(* CODESYS project mobject-server.library
   Company: mobject
   DefaultNamespace: mobject-server
   Version: 0.10.0
   Placeholder: mobject-server
   Author: mobject dev team
   Title: mobject-server

Project tree, tasks and I/O mapping:
  libraries: mobject-core, 0.3.0 (mobject); Tc2_Standard, * (Beckhoff Automation GmbH); Tc2_System, * (Beckhoff Automation GmbH); Tc2_Utilities, * (Beckhoff Automation GmbH)
  _Internal/
    AsyncResponse/
      HeaderAccessor/
        interface I_AsyncResponseHeaderAccessor: TryGetResponseIdFromRequest, TryGetSessionIdFromRequest, TryGetSessionIdFromResponse
      Manager/
        function block AsyncResponseManager [ST]: FB_init, CreateAsyncResponseSessionData, CreateAsyncResponseSessionDataProxy, TryConvertResponseToAsyncResponseSessionData, TryHandleIncomingRequest
        interface I_AsyncResponseManager: TryConvertResponseToAsyncResponseSessionData, TryHandleIncomingRequest
      Middleware/
        function block AsyncResponseMiddleware [ST]: FB_init, Handle
      Proxy/
        function block AsyncResponseSessionDataProxy [ST]: FB_init, TryGetAsyncResponseSessionData, Error, IsPending, Success, SuccessWithPayload, SuggestedRetryDelayInMs, TryUpdateServerResponse
      SessionData/
        function block AsyncResponseSessionData [ST]: FB_init, FB_exit, CopyPayloadData, DeletePayloadData, Error, IsPending, Success, SuccessWithPayload, SuggestedRetryDelayInMs, TryUpdateServerResponse
        interface I_AsyncResponseSessionData: Error, IsPending, Success, SuccessWithPayload, SuggestedRetryDelayInMs, TryUpdateServerResponse
    ChunkedRequests/
      ChunkedRequest/
        function block ChunkedRequest [ST]: FB_init, CreatedTimestamp, Header, PayloadAddress, PayloadSizeInBytes
      HeaderAccessor/
        interface I_ChunkedRequestsHeaderAccessor: TryGetChunkSequenceFromRequest, TryGetChunkTotalFromRequest, TryGetHasMoreChunksFromRequest, TryGetRequestIdFromRequest, TryGetSessionIdFromRequest
      Manager/
        function block ChunkedRequestsManager [ST]: FB_init, CreateChunkedRequestData, TryHandleIncomingRequest
        interface I_ChunkedRequestsManager: TryHandleIncomingRequest
      Middleware/
        function block ChunkedRequestsMiddleware [ST]: FB_init, Handle
      SessionData/
        function block ChunkedRequestData [ST]: FB_init, FB_exit, CreateBuffer, DestroyBuffer, IsComplete, PayloadAddress, PayloadSizeInBytes, TryAddChunkedPayload
        interface I_ChunkedRequestData: IsComplete, PayloadAddress, PayloadSizeInBytes, TryAddChunkedPayload
    ChunkedResponses/
      HeaderAccessor/
        interface I_ChunkedResponseHeaderAccessor: TryGetResponseIdFromRequest, TryGetSessionIdFromRequest, TryGetSessionIdFromResponse, UpdateResponseWithHasMoreChunks
      Manager/
        function block ChunkedResponseManager [ST]: FB_init, CreateChunkedResponseData, HandleSuccessWithPayload, TryHandleIncomingRequest
        interface I_ChunkedResponseManager: HandleSuccessWithPayload, TryHandleIncomingRequest
      Middleware/
        function block ChunkedResponsesMiddleware [ST]: FB_init, Handle
      ServerResponse/
        function block ChunkableServerResponse [ST]: FB_init, Accepted, Busy, Error, Header, HeadersSent, Pending, Success, SuccessWithPayload
      SessionData/
        function block ChunkedResponseData [ST]: FB_init, FB_exit, StoreData, SendComplete, SendNextChunk, SizeRemaining
        interface I_ChunkedResponseData: SendComplete, SendNextChunk, SizeRemaining
    Header/
      function block Header [ST]: FB_init, FB_exit, ToString, TryGetField, TryWriteField
      interface I_Header: ToString, TryGetField, TryWriteField
    HeaderAccessor/
      function block HeaderAccessor [ST]: ContentType_Json, HeaderKey_Accept, HeaderKey_ChunkSequence, HeaderKey_ChunkTotal, HeaderKey_ContentType, HeaderKey_HasMoreChunks, HeaderKey_Message, HeaderKey_MethodName, HeaderKey_RequestId, HeaderKey_ResponseId, HeaderKey_RetryDelay, HeaderKey_SessionId, HeaderKey_Status, HeaderKey_Type, StatusValue_Accepted, StatusValue_Busy, StatusValue_Error, StatusValue_Pending, StatusValue_Success, TryGetAcceptResponseFormatFromRequest, TryGetChunkSequenceFromRequest, TryGetChunkTotalFromRequest, TryGetContentTypeFromRequest, TryGetHasMoreChunksFromRequest, TryGetMethodNameFromRequest, TryGetRequestIdFromRequest, TryGetResponseIdFromRequest, TryGetSessionIdFromRequest, TryGetSessionIdFromResponse, TryGetTypeFromRequest, UpdateRequestWithSessionId, UpdateResponseWithAccepted, UpdateResponseWithBusy, UpdateResponseWithError, UpdateResponseWithHasMoreChunks, UpdateResponseWithPending, UpdateResponseWithSessionId, UpdateResponseWithSuccess
    Middleware/
      Base/
        function block MiddlewareBase [ST]: Next, Handle, NextMiddleware
      Interface/
        interface I_Middleware: Handle, NextMiddleware
      Stack/
        function block MiddlewareStack [ST]: Handle, Use
    Request/
      Interface/
        interface I_Request: CreatedTimestamp, Header, PayloadAddress, PayloadSizeInBytes
      function block Request [ST]: FB_init, CreatedTimestamp, Header, PayloadAddress, PayloadSizeInBytes
    ResponseId/
      Interface/
        interface I_ResponseIdGenerator: Generate
      function block SequentialResponseIdGenerator [ST]: Generate
    RPC/
      AsyncRpcCall/
        function block AsyncRpcCall [ST]: FB_init, FB_exit, Call
        interface I_AsyncRpcCall: Call
      AsyncRpcCallQueue/
        function block AsyncRpcCallQueue [ST]: FB_exit, CreateCall, DisposeAll, CyclicCall, TryAddRpcCall
        interface I_AsyncRpcCallQueue: TryAddRpcCall
      Handlers/
        function block AsynchronousRpcHandlers [ST]: HasHandlers, RegisterHandler, TryGetByMethodName
        interface I_AsynchronousRpcHandlers: HasHandlers, TryGetByMethodName
        interface I_HostAsynchronousRpcHandlers: RegisterHandler
        interface I_HostSynchronousRpcHandlers: RegisterHandler
        interface I_SynchronousRpcHandlers: HasHandlers, TryGetByMethodName
        function block SynchronousRpcHandlers [ST]: HasHandlers, RegisterHandler, TryGetByMethodName
      HeaderAccessor/
        interface I_RpcHeaderAccessor: ContentType_Json, TryGetAcceptResponseFormatFromRequest, TryGetContentTypeFromRequest, TryGetMethodNameFromRequest, TryGetTypeFromRequest
      Manager/
        interface I_RpcManager: TryHandleIncomingRequest
        function block RpcManager [ST]: FB_init, HandleAsyncRpcRequest, HandleSyncRpcRequest, TryCreateAsynchronousRpcResponse, TryCreateDeserializer, TryCreateSerializer, TryCreateSynchronousRpcResponse, TryHandleIncomingRequest
      Middleware/
        function block RpcMiddleware [ST]: FB_init, Handle
      RegisteredRpcApis/
        function block RegisteredRpcApis [ST]: FB_exit, CreateEnumerator, CyclicCall, HasRegisteredRpcApis, RegisterRpcApi
      Response/
        Async/
          function block AsynchronousRpcResponse [ST]: FB_init, FB_exit, SendSuccessResponseUsingSeralizer, CompleteWithBase64, CompleteWithBool, CompleteWithBytesAsHex, CompleteWithDateTime, CompleteWithDcTime, CompleteWithDint, CompleteWithFileTime, CompleteWithLint, CompleteWithLreal, CompleteWithNull, CompleteWithObject, CompleteWithReal, CompleteWithSerializer, CompleteWithString, CompleteWithUdint, CompleteWithUlint, GetSerializer, RejectWithMessage
          interface I_AsynchronousRpcResponse: CompleteWithBase64, CompleteWithBool, CompleteWithBytesAsHex, CompleteWithDateTime, CompleteWithDcTime, CompleteWithDint, CompleteWithFileTime, CompleteWithLint, CompleteWithLreal, CompleteWithNull, CompleteWithObject, CompleteWithReal, CompleteWithSerializer, CompleteWithString, CompleteWithUdint, CompleteWithUlint, GetSerializer, RejectWithMessage
        Factory/
          function block AsynchronousRpcResponseFactory [ST]: FB_init, TryCreate
          interface I_AsynchronousRpcResponseFactory: TryCreate
        Sync/
          interface I_SynchronousRpcResponse: CompleteWithBase64, CompleteWithBool, CompleteWithBytesAsHex, CompleteWithDateTime, CompleteWithDcTime, CompleteWithDint, CompleteWithFileTime, CompleteWithLint, CompleteWithLreal, CompleteWithNull, CompleteWithObject, CompleteWithReal, CompleteWithSerializer, CompleteWithString, CompleteWithUdint, CompleteWithUlint, GetSerializer, RejectWithMessage, TryMakeAsynchronous
          function block SynchronousRpcResponse [ST]: FB_init, FB_exit, SendSuccessResponseUsingSeralizer, CompleteWithBase64, CompleteWithBool, CompleteWithBytesAsHex, CompleteWithDateTime, CompleteWithDcTime, CompleteWithDint, CompleteWithFileTime, CompleteWithLint, CompleteWithLreal, CompleteWithNull, CompleteWithObject, CompleteWithReal, CompleteWithSerializer, CompleteWithString, CompleteWithUdint, CompleteWithUlint, GetSerializer, RejectWithMessage, TryMakeAsynchronous
    ServerResponse/
      Data/
        data type ResponseData
      HeaderAccessor/
        interface I_ServerResponseHeaderAccessor: UpdateResponseWithAccepted, UpdateResponseWithBusy, UpdateResponseWithError, UpdateResponseWithPending, UpdateResponseWithSuccess
      Interface/
        interface I_ServerResponse: Accepted, Busy, Error, Header, HeadersSent, Pending, Success, SuccessWithPayload
      function block ServerResponse [ST]: FB_init, CompleteResponseWithoutPayload, CompleteResponseWithPayload, Accepted, Busy, Error, Header, HeadersSent, Pending, Success, SuccessWithPayload, TryGetData
    Sessions/
      HeaderAccessor/
        interface I_SessionHeaderAccessor: TryGetSessionIdFromRequest, UpdateRequestWithSessionId, UpdateResponseWithSessionId
      Manager/
        interface I_SessionManager: CreateSession, DisposeAllSessions, IsValidSession, RefreshSession
        function block SessionManager [ST]: FB_init, FB_exit, CheckForExpiredSessions, CreateNewSession, CreateSession, CyclicCall, DisposeAllSessions, DisposeSession, DisposeSessionDataById, IsValidSession, RefreshSession, SessionCount, TryRetreiveSessionDataById, TryStoreSessionDataById
      Middleware/
        function block SessionsMiddleware [ST]: FB_init, Handle
      Session/
        interface I_Session: AddOrUpdateStorage, DisposeAllDataFromStorage, DisposeDataFromStorage, Id, LastAccessedTimestamp, Refresh, TryGetDataFromStorage
        function block Session [ST]: FB_init, FB_exit, AddOrUpdateStorage, DisposeAllDataFromStorage, DisposeDataFromStorage, Id, LastAccessedTimestamp, Refresh, TryGetDataFromStorage
      SessionData/
        interface I_SessionData
      SessionId/
        interface I_SessionIdGenerator: Generate
        function block SequentialSessionIdGenerator [ST]: Generate
      Storage/
        interface I_SessionStorage: DisposeSessionDataById, TryRetreiveSessionDataById, TryStoreSessionDataById
    TimeStamp/
      interface I_Timestamp: IsDurationElapsed, TimeSince
      function block SystemTimestamp [ST]: FB_init, IsDurationElapsed, SetNow, TimeSince
  GVLs/
    global variables ServerConfiguration
  RpcApi/
    interface I_RpcApi: CyclicCall, RegisterAsynchronousRpcHandlersWith, RegisterSynchronousRpcHandlersWith
  RpcHandler/
    Examples/
      function block AsyncConcatStringRpcHandler [ST]: Handle
      function block ConcatStringRpcHandler [ST]: Handle
    interface I_AsynchronousRpcHandler: Handle
    interface I_SynchronousRpcHandler: Handle
  RpcServer/
    interface I_RpcServer: RegisterApi, RegisterAsynchronousRpcHandler, RegisterSynchronousRpcHandler
    function block RpcServer [ST]: FB_init, CyclicCall, HandleRequest, RegisterApi, RegisterAsynchronousRpcHandler, RegisterSynchronousRpcHandler, SessionCount, Use
*)

// _Internal/ServerResponse/Data/ResponseData
TYPE ResponseData : 
STRUCT
	Header : STRING(ServerConfiguration.HEADER_STRING_SIZE);
	Payload : STRING(ServerConfiguration.PAYLOAD_STRING_SIZE);
END_STRUCT
END_TYPE

// GVLs/ServerConfiguration
{attribute 'qualified_only'}
VAR_GLOBAL CONSTANT
	HEADER_STRING_SIZE : UDINT := 1024; 
	PAYLOAD_STRING_SIZE : UDINT := 8000; // typically 1/8th of the Runtime Stack Size
END_VAR

// _Internal/AsyncResponse/HeaderAccessor/I_AsyncResponseHeaderAccessor
INTERFACE I_AsyncResponseHeaderAccessor

METHOD PUBLIC TryGetResponseIdFromRequest : BOOL
VAR_INPUT
	Request : I_Request;
	Destination : ANY;
END_VAR
END_METHOD

METHOD PUBLIC TryGetSessionIdFromRequest : BOOL
VAR_INPUT
	Request : I_Request;
	Destination : REFERENCE TO T_MAXSTRING;
END_VAR
END_METHOD

METHOD PUBLIC TryGetSessionIdFromResponse : BOOL
VAR_INPUT
	Response : I_ServerResponse;
	Destination : ANY;
END_VAR
END_METHOD

END_INTERFACE

// _Internal/Request/Request
{attribute 'linkalways'} 
{attribute 'no_explicit_call' := 'This FB is a CLASS and must be accessed using methods or properties'}
{attribute 'enable_dynamic_creation'}
FUNCTION_BLOCK Request Extends Disposable IMPLEMENTS I_Request
VAR
	_header : I_Header;
	_payloadAddress : POINTER TO STRING(0);
	_payloadSizeInBytes : UDINT;	
	_createdTimestamp : SystemTimestamp;
END_VAR

METHOD FB_init : BOOL
VAR_INPUT
	bInitRetains : BOOL; // if TRUE, the retain variables are initialized (warm start / cold start)
	bInCopyCode : BOOL;  // if TRUE, the instance afterwards gets moved into the copy code (online change)
	Header : I_Header;
	Payload : ANY_STRING;
END_VAR
_header := Header;
_payloadSizeInBytes := DINT_TO_UDINT(Payload.diSize);
_payloadAddress := Payload.pValue;
END_METHOD

PROPERTY PUBLIC CreatedTimestamp : I_Timestamp
GET
CreatedTimestamp := _createdTimestamp;
END_GET
END_PROPERTY

PROPERTY PUBLIC Header : I_Header
GET
Header := _header;
END_GET
END_PROPERTY

PROPERTY PUBLIC PayloadAddress : POINTER TO STRING
GET
PayloadAddress := _payloadAddress;
END_GET
END_PROPERTY

PROPERTY PUBLIC PayloadSizeInBytes : UDINT
GET
PayloadSizeInBytes := _payloadSizeInBytes;
END_GET
END_PROPERTY

END_FUNCTION_BLOCK

// _Internal/Request/Interface/I_Request
INTERFACE I_Request EXTENDS I_Disposable

PROPERTY PUBLIC CreatedTimestamp : I_Timestamp
GET
END_GET
END_PROPERTY

PROPERTY PUBLIC Header : I_Header
GET
END_GET
END_PROPERTY

PROPERTY PUBLIC PayloadAddress : POINTER TO STRING
GET
END_GET
END_PROPERTY

PROPERTY PUBLIC PayloadSizeInBytes : UDINT
GET
END_GET
END_PROPERTY

END_INTERFACE

// _Internal/TimeStamp/I_Timestamp
INTERFACE I_Timestamp

METHOD PUBLIC IsDurationElapsed : BOOL
VAR_INPUT
	Duration : TIME;
END_VAR
END_METHOD

PROPERTY PUBLIC TimeSince : TIME
GET
END_GET
END_PROPERTY

END_INTERFACE

// _Internal/Header/Header
{attribute 'linkalways'} 
{attribute 'no_explicit_call' := 'This FB is a CLASS and must be accessed using methods or properties'}
{attribute 'enable_dynamic_creation'}
FUNCTION_BLOCK Header IMPLEMENTS I_Header
VAR
	jsonParser : JsonDomParser;
END_VAR

METHOD FB_init : BOOL
VAR_INPUT
	bInitRetains : BOOL; // if TRUE, the retain variables are initialized (warm start / cold start)
	bInCopyCode : BOOL;  // if TRUE, the instance afterwards gets moved into the copy code (online change)
	InitialHeader : REFERENCE TO STRING(ServerConfiguration.HEADER_STRING_SIZE);
END_VAR
VAR
	root : SJsonValue;
END_VAR
IF __ISVALIDREF(InitialHeader) THEN
	root := jsonParser.ParseDocument(InitialHeader);
ELSE
	root := jsonParser.NewDocument();
	jsonParser.SetObject(root);
END_IF
END_METHOD

METHOD FB_exit : BOOL
VAR_INPUT
	bInCopyCode : BOOL; // if TRUE, the exit method is called for exiting an instance that is copied afterwards (online change).
END_VAR
IF bInCopyCode THEN
	RETURN;
END_IF

jsonParser.NewDocument();
END_METHOD

METHOD PUBLIC ToString
VAR_INPUT
	Destination : REFERENCE TO STRING(ServerConfiguration.HEADER_STRING_SIZE);
END_VAR
jsonParser.CopyDocument(Destination,sizeof(Destination));
END_METHOD

METHOD PUBLIC TryGetField : BOOL;
VAR_INPUT
	Key : STRING;
	Destination : ANY;
END_VAR
IF Key = '' THEN
	RETURN;
END_IF

TryGetField := jsonParser.TryRead(Key, Destination);
END_METHOD

METHOD PUBLIC TryWriteField : BOOL;
VAR_INPUT
	Key : STRING;
	Source : ANY;
END_VAR
IF Key = '' THEN
	RETURN;
END_IF

TryWriteField := jsonParser.TryWrite(Key, Source);
END_METHOD

END_FUNCTION_BLOCK

// _Internal/Header/I_Header
INTERFACE I_Header

METHOD PUBLIC ToString
VAR_INPUT
	Destination : REFERENCE TO STRING(ServerConfiguration.HEADER_STRING_SIZE);
END_VAR
END_METHOD

METHOD PUBLIC TryGetField : BOOL;
VAR_INPUT
	Key : STRING;
	Destination : ANY;
END_VAR
END_METHOD

METHOD PUBLIC TryWriteField : BOOL;
VAR_INPUT
	Key : STRING;
	Source : ANY;
END_VAR
END_METHOD

END_INTERFACE

// _Internal/TimeStamp/SystemTimestamp
FUNCTION_BLOCK SystemTimestamp Implements I_Timestamp
VAR
	recordedTime : ULINT;
END_VAR

METHOD FB_init : BOOL
VAR_INPUT
	bInitRetains : BOOL; // if TRUE, the retain variables are initialized (warm start / cold start)
	bInCopyCode : BOOL;  // if TRUE, the instance afterwards gets moved into the copy code (online change)
END_VAR
SetNow();
END_METHOD

METHOD PUBLIC IsDurationElapsed : BOOL
VAR_INPUT
	Duration : TIME;
END_VAR
VAR
	currentTime : ULINT;
	elapsedDuration : ULINT;
	durationInHundredNs : ULINT;
END_VAR
currentTime := F_GetSystemTime();

// Convert duration from milliseconds to 100-nanosecond intervals.
// Since 1 ms = 10,000 * 100 ns.
durationInHundredNs := TIME_TO_ULINT(duration) * 10000; 

// Calculate the time that must elapse before the timestamp is considered 'expired'.
elapsedDuration := recordedTime + durationInHundredNs;

// Check if the current time is beyond the elapsed duration.
IsDurationElapsed := currentTime > elapsedDuration;
END_METHOD

METHOD PUBLIC SetNow
VAR_INPUT
END_VAR
recordedTime := F_GetSystemTime();
END_METHOD

PROPERTY PUBLIC TimeSince : TIME
GET
VAR
	currentTime : ULINT;
	elapsedDurationInHundredNs : ULINT;
	convertTime : ULINT;
END_VAR
currentTime := F_GetSystemTime();

elapsedDurationInHundredNs := currentTime - recordedTime;
convertTime := elapsedDurationInHundredNs / 10000;
TimeSince := ULINT_TO_TIME(convertTime);
END_GET
END_PROPERTY

END_FUNCTION_BLOCK

// _Internal/ServerResponse/Interface/I_ServerResponse
INTERFACE I_ServerResponse

METHOD PUBLIC Accepted
VAR_INPUT
END_VAR
END_METHOD

METHOD PUBLIC Busy
VAR_INPUT
END_VAR
END_METHOD

METHOD PUBLIC Error
VAR_INPUT
	Message : T_MAXSTRING;
END_VAR
END_METHOD

PROPERTY PUBLIC Header : I_Header
GET
END_GET
END_PROPERTY

PROPERTY PUBLIC HeadersSent : BOOL
GET
END_GET
END_PROPERTY

METHOD PUBLIC Pending
VAR_INPUT
	ResponseId : REFERENCE TO T_MAXSTRING;
	RetryDelayInMs : UDINT;
END_VAR
END_METHOD

METHOD PUBLIC Success
VAR_INPUT
END_VAR
END_METHOD

METHOD PUBLIC SuccessWithPayload
VAR_INPUT
	PayloadDataAddress : PVOID;
	PayloadDataSize : UDINT;
END_VAR
END_METHOD

END_INTERFACE

// _Internal/AsyncResponse/Manager/AsyncResponseManager
{attribute 'linkalways'} 
{attribute 'no_explicit_call' := 'This FB is a CLASS and must be accessed using methods or properties'}
{attribute 'enable_dynamic_creation'}
FUNCTION_BLOCK AsyncResponseManager IMPLEMENTS I_AsyncResponseManager
VAR
	sessionStorage : I_SessionStorage;
	responseIdGenerator : I_ResponseIdGenerator;
	headerAccessor : I_AsyncResponseHeaderAccessor;
END_VAR

METHOD FB_init : BOOL
VAR_INPUT
	bInitRetains : BOOL; // if TRUE, the retain variables are initialized (warm start / cold start)
	bInCopyCode : BOOL;  // if TRUE, the instance afterwards gets moved into the copy code (online change)
	SessionStorage : I_SessionStorage;
	ResponseIdGenerator : I_ResponseIdGenerator;
	HeaderAccessor : I_AsyncResponseHeaderAccessor;
END_VAR
THIS^.sessionStorage := SessionStorage;
THIS^.responseIdGenerator := ResponseIdGenerator;
THIS^.headerAccessor := HeaderAccessor;
END_METHOD

METHOD PROTECTED CreateAsyncResponseSessionData : I_AsyncResponseSessionData
VAR_INPUT
	RetryDelayInMs : UDINT;
END_VAR
VAR
	pAsyncResponseSessionData : POINTER TO AsyncResponseSessionData;
END_VAR
pAsyncResponseSessionData := __NEW(AsyncResponseSessionData(SuggestedRetryDelayInMs := RetryDelayInMs));
CreateAsyncResponseSessionData := pAsyncResponseSessionData^;
END_METHOD

METHOD PROTECTED CreateAsyncResponseSessionDataProxy : I_AsyncResponseSessionData
VAR_INPUT
	ProxySessionId : T_MAXSTRING;
	ProxyResponseId : T_MAXSTRING;
END_VAR
VAR
	pAsyncResponseSessionDataProxy : POINTER TO AsyncResponseSessionDataProxy;
END_VAR
pAsyncResponseSessionDataProxy := __NEW(AsyncResponseSessionDataProxy(SessionStorage := THIS^.sessionStorage, SessionId := ProxySessionId, ResponseId := ProxyResponseId));
CreateAsyncResponseSessionDataProxy := pAsyncResponseSessionDataProxy^;
END_METHOD

METHOD TryConvertResponseToAsyncResponseSessionData : BOOL
VAR_INPUT
	Response : I_ServerResponse;
	RetryDelayInMs : UDINT;
	Destination : REFERENCE TO I_AsyncResponseSessionData;
END_VAR
VAR
	sessionId : T_MAXSTRING;
	responseId : T_MAXSTRING;
	newResponseId : T_MAXSTRING;
	asyncResponseSessionData : I_AsyncResponseSessionData;
END_VAR
IF NOT headerAccessor.TryGetSessionIdFromResponse(Response,sessionId) THEN
	Response.Error('Unable to create a pending response without a sessionId');
	RETURN;
END_IF

asyncResponseSessionData := CreateAsyncResponseSessionData(RetryDelayInMs);
responseId := responseIdGenerator.Generate();

IF NOT sessionStorage.TryStoreSessionDataById(sessionId, responseId, asyncResponseSessionData) THEN
	Response.Error('Unable to store pending response');
	asyncResponseSessionData.Dispose();
	RETURN;
END_IF

Response.Pending(responseId, RetryDelayInMs);
Destination := CreateAsyncResponseSessionDataProxy(sessionId, responseId);
TryConvertResponseToAsyncResponseSessionData := true;
END_METHOD

METHOD PUBLIC TryHandleIncomingRequest : BOOL
VAR_INPUT
	Request : I_Request;
	Response : I_ServerResponse;
END_VAR
VAR
	responseId : T_MAXSTRING;
	sessionId : T_MAXSTRING;
	sessionData : I_SessionData;
	asyncResponseData : I_AsyncResponseSessionData;
END_VAR
IF NOT headerAccessor.TryGetResponseIdFromRequest(Request, responseId) THEN
	RETURN;
END_IF

IF NOT headerAccessor.TryGetSessionIdFromRequest(Request, sessionId) THEN
	RETURN;
END_IF

IF NOT sessionStorage.TryRetreiveSessionDataById(sessionId, responseId, sessionData) THEN
	RETURN;
END_IF

IF NOT __QUERYINTERFACE(sessionData, asyncResponseData) THEN
	RETURN;
END_IF

IF asyncResponseData.IsPending THEN
	Response.Pending(responseId, asyncResponseData.SuggestedRetryDelayInMs);
	TryHandleIncomingRequest := TRUE;
	RETURN;
END_IF

IF NOT asyncResponseData.TryUpdateServerResponse(Response) THEN	
	Response.Error('Unable to update server response with pending data');
	TryHandleIncomingRequest := TRUE;
	RETURN;
END_IF

sessionStorage.DisposeSessionDataById(sessionId, responseId);
TryHandleIncomingRequest := TRUE;
END_METHOD

END_FUNCTION_BLOCK

// _Internal/AsyncResponse/Manager/I_AsyncResponseManager
INTERFACE I_AsyncResponseManager

METHOD TryConvertResponseToAsyncResponseSessionData : BOOL
VAR_INPUT
	Response : I_ServerResponse;
	RetryDelayInMs : UDINT;
	Destination : REFERENCE TO I_AsyncResponseSessionData;
END_VAR
END_METHOD

METHOD PUBLIC TryHandleIncomingRequest : BOOL
VAR_INPUT
	Request : I_Request;
	Response : I_ServerResponse;
END_VAR
END_METHOD

END_INTERFACE

// _Internal/AsyncResponse/SessionData/I_AsyncResponseSessionData
INTERFACE I_AsyncResponseSessionData EXTENDS I_SessionData

METHOD PUBLIC Error
VAR_INPUT
	Message : T_MAXSTRING;
END_VAR
END_METHOD

PROPERTY PUBLIC IsPending : BOOL
GET
END_GET
END_PROPERTY

METHOD PUBLIC Success
VAR_INPUT
END_VAR
END_METHOD

METHOD PUBLIC SuccessWithPayload
VAR_INPUT
	PayloadDataAddress : PVOID;
	PayloadDataSize : UDINT;
END_VAR
END_METHOD

PROPERTY PUBLIC SuggestedRetryDelayInMs : UDINT
GET
END_GET
SET
END_SET
END_PROPERTY

METHOD PUBLIC TryUpdateServerResponse : BOOL
VAR_INPUT
	Response : I_ServerResponse;
END_VAR
END_METHOD

END_INTERFACE

// _Internal/Sessions/SessionData/I_SessionData
INTERFACE I_SessionData EXTENDS I_Disposable

END_INTERFACE

// _Internal/Sessions/Storage/I_SessionStorage
INTERFACE I_SessionStorage

METHOD PUBLIC DisposeSessionDataById
VAR_INPUT
	SessionId : T_MAXSTRING;
	StorageId : T_MAXSTRING;
END_VAR
END_METHOD

METHOD PUBLIC TryRetreiveSessionDataById : BOOL
VAR_INPUT
	SessionId : T_MAXSTRING;
	StorageId : T_MAXSTRING;
	Destination : REFERENCE TO I_SessionData;
END_VAR
END_METHOD

METHOD PUBLIC TryStoreSessionDataById : BOOL
VAR_INPUT
	SessionId : T_MAXSTRING;
	StorageId : T_MAXSTRING;
	Source : I_SessionData;
END_VAR
END_METHOD

END_INTERFACE

// _Internal/ResponseId/Interface/I_ResponseIdGenerator
INTERFACE I_ResponseIdGenerator

METHOD PUBLIC Generate : T_MAXSTRING
VAR_INPUT
END_VAR
END_METHOD

END_INTERFACE

// _Internal/HeaderAccessor/HeaderAccessor
FUNCTION_BLOCK HeaderAccessor IMPLEMENTS I_SessionHeaderAccessor, I_ServerResponseHeaderAccessor, I_AsyncResponseHeaderAccessor, I_ChunkedResponseHeaderAccessor, I_ChunkedRequestsHeaderAccessor, I_RpcHeaderAccessor

PROPERTY PUBLIC ContentType_Json : T_MAXSTRING
GET
ContentType_Json := 'application/json';
END_GET
SET
// must keep so that it works with ANY
END_SET
END_PROPERTY

PROPERTY PUBLIC HeaderKey_Accept : T_MAXSTRING
GET
HeaderKey_Accept := 'Accept';
END_GET
SET
// must keep so that it works with ANY
END_SET
END_PROPERTY

PROPERTY PUBLIC HeaderKey_ChunkSequence : T_MAXSTRING
GET
HeaderKey_ChunkSequence := 'Chunk-Sequence';
END_GET
SET
// must keep so that it works with ANY
END_SET
END_PROPERTY

PROPERTY PUBLIC HeaderKey_ChunkTotal : T_MAXSTRING
GET
HeaderKey_ChunkTotal := 'Chunk-Total';
END_GET
SET
// must keep so that it works with ANY
END_SET
END_PROPERTY

PROPERTY PUBLIC HeaderKey_ContentType : T_MAXSTRING
GET
HeaderKey_ContentType := 'Content-Type';
END_GET
SET
// must keep so that it works with ANY
END_SET
END_PROPERTY

PROPERTY PUBLIC HeaderKey_HasMoreChunks : T_MAXSTRING
GET
HeaderKey_HasMoreChunks := 'Has-More-Chunks';
END_GET
SET
// must keep so that it works with ANY
END_SET
END_PROPERTY

PROPERTY PUBLIC HeaderKey_Message : T_MAXSTRING
GET
HeaderKey_Message := 'Message';
END_GET
SET
// must keep so that it works with ANY
END_SET
END_PROPERTY

PROPERTY PUBLIC HeaderKey_MethodName : T_MAXSTRING
GET
HeaderKey_MethodName := 'Method-Name';
END_GET
SET
// must keep so that it works with ANY
END_SET
END_PROPERTY

PROPERTY PUBLIC HeaderKey_RequestId : T_MAXSTRING
GET
HeaderKey_RequestId := 'Request-Id';
END_GET
SET
// must keep so that it works with ANY
END_SET
END_PROPERTY

PROPERTY PUBLIC HeaderKey_ResponseId : T_MAXSTRING
GET
HeaderKey_ResponseId := 'Response-Id';
END_GET
SET
// must keep so that it works with ANY
END_SET
END_PROPERTY

PROPERTY PUBLIC HeaderKey_RetryDelay : T_MAXSTRING
GET
HeaderKey_RetryDelay := 'Retry-Delay';
END_GET
SET
// must keep so that it works with ANY
END_SET
END_PROPERTY

PROPERTY PUBLIC HeaderKey_SessionId : T_MAXSTRING
GET
HeaderKey_SessionId := 'Session-Id';
END_GET
SET
// must keep so that it works with ANY
END_SET
END_PROPERTY

PROPERTY PUBLIC HeaderKey_Status : T_MAXSTRING
GET
HeaderKey_Status := 'Status';
END_GET
SET
// must keep so that it works with ANY
END_SET
END_PROPERTY

PROPERTY PUBLIC HeaderKey_Type : T_MAXSTRING
GET
HeaderKey_Type := 'Type';
END_GET
SET
// must keep so that it works with ANY
END_SET
END_PROPERTY

PROPERTY PUBLIC StatusValue_Accepted : T_MAXSTRING
GET
StatusValue_Accepted := 'Accepted';
END_GET
SET
// must keep so that it works with ANY
END_SET
END_PROPERTY

PROPERTY PUBLIC StatusValue_Busy : T_MAXSTRING
GET
StatusValue_Busy := 'Busy';
END_GET
SET
// must keep so that it works with ANY
END_SET
END_PROPERTY

PROPERTY PUBLIC StatusValue_Error : T_MAXSTRING
GET
StatusValue_Error := 'Error';
END_GET
SET
// must keep so that it works with ANY
END_SET
END_PROPERTY

PROPERTY PUBLIC StatusValue_Pending : T_MAXSTRING
GET
StatusValue_Pending := 'Pending';
END_GET
SET
// must keep so that it works with ANY
END_SET
END_PROPERTY

PROPERTY PUBLIC StatusValue_Success : T_MAXSTRING
GET
StatusValue_Success := 'Success';
END_GET
SET
// must keep so that it works with ANY
END_SET
END_PROPERTY

METHOD PUBLIC TryGetAcceptResponseFormatFromRequest : BOOL
VAR_INPUT
	Request : I_Request;
	Destination : ANY;
END_VAR
TryGetAcceptResponseFormatFromRequest := Request.Header.TryGetField(HeaderKey_Accept,Destination);
END_METHOD

METHOD PUBLIC TryGetChunkSequenceFromRequest : BOOL
VAR_INPUT
	Request : I_Request;
	Destination : REFERENCE TO DINT;
END_VAR
VAR
	chunkSequence : DINT;
END_VAR
IF NOT Request.Header.TryGetField(HeaderKey_ChunkSequence,chunkSequence) THEN
	RETURN;
END_IF

Destination := chunkSequence;
TryGetChunkSequenceFromRequest := TRUE;
END_METHOD

METHOD PUBLIC TryGetChunkTotalFromRequest : BOOL
VAR_INPUT
	Request : I_Request;
	Destination : REFERENCE TO DINT;
END_VAR
VAR
	chunkTotal : DINT;
END_VAR
IF NOT Request.Header.TryGetField(HeaderKey_ChunkTotal,chunkTotal) THEN
	RETURN;
END_IF

Destination := chunkTotal;
TryGetChunkTotalFromRequest := TRUE;
END_METHOD

METHOD PUBLIC TryGetContentTypeFromRequest : BOOL
VAR_INPUT
	Request : I_Request;
	Destination : ANY;
END_VAR
TryGetContentTypeFromRequest := Request.Header.TryGetField(HeaderKey_ContentType,Destination);
END_METHOD

METHOD PUBLIC TryGetHasMoreChunksFromRequest : BOOL
VAR_INPUT
	Request : I_Request;
	Destination : REFERENCE TO BOOL;
END_VAR
VAR
	hasMoreChunks : BOOL;
END_VAR
IF NOT Request.Header.TryGetField(HeaderKey_HasMoreChunks,hasMoreChunks) THEN
	RETURN;
END_IF

Destination := hasMoreChunks;
TryGetHasMoreChunksFromRequest := TRUE;
END_METHOD

METHOD PUBLIC TryGetMethodNameFromRequest : BOOL
VAR_INPUT
	Request : I_Request;
	Destination : ANY;
END_VAR
TryGetMethodNameFromRequest := Request.Header.TryGetField(HeaderKey_MethodName,Destination);
END_METHOD

METHOD PUBLIC TryGetRequestIdFromRequest : BOOL
VAR_INPUT
	Request : I_Request;
	Destination : REFERENCE TO T_MAXSTRING;
END_VAR
VAR
	requestId : T_MAXSTRING;
END_VAR
IF NOT Request.Header.TryGetField(HeaderKey_RequestId,requestId) THEN
	RETURN;
END_IF

Destination := requestId;
TryGetRequestIdFromRequest := TRUE;
END_METHOD

METHOD PUBLIC TryGetResponseIdFromRequest : BOOL
VAR_INPUT
	Request : I_Request;
	Destination : ANY;
END_VAR
TryGetResponseIdFromRequest := Request.Header.TryGetField(HeaderKey_ResponseId,Destination);
END_METHOD

METHOD PUBLIC TryGetSessionIdFromRequest : BOOL
VAR_INPUT
	Request : I_Request;
	Destination : REFERENCE TO T_MAXSTRING;
END_VAR
VAR
	sessionId : T_MAXSTRING;
END_VAR
IF NOT Request.Header.TryGetField(HeaderKey_SessionId, sessionId) THEN
	RETURN;
END_IF

Destination := sessionId;
TryGetSessionIdFromRequest := TRUE;
END_METHOD

METHOD PUBLIC TryGetSessionIdFromResponse : BOOL
VAR_INPUT
	Response : I_ServerResponse;
	Destination : ANY;
END_VAR
TryGetSessionIdFromResponse := Response.Header.TryGetField(HeaderKey_SessionId,Destination);
END_METHOD

METHOD PUBLIC TryGetTypeFromRequest : BOOL
VAR_INPUT
	Request : I_Request;
	Destination : ANY;
END_VAR
TryGetTypeFromRequest := Request.Header.TryGetField(HeaderKey_Type,Destination);
END_METHOD

METHOD PUBLIC UpdateRequestWithSessionId
VAR_INPUT
	Request : I_Request;
	SessionId : T_MAXSTRING;
END_VAR
Request.Header.TryWriteField(HeaderKey_SessionId,SessionId);
END_METHOD

METHOD PUBLIC UpdateResponseWithAccepted
VAR_INPUT
	Response : I_ServerResponse;
END_VAR
Response.Header.TryWriteField(HeaderKey_Status,StatusValue_Accepted);
END_METHOD

METHOD PUBLIC UpdateResponseWithBusy
VAR_INPUT
	Response : I_ServerResponse;
END_VAR
Response.Header.TryWriteField(HeaderKey_Status,StatusValue_Busy);
END_METHOD

METHOD PUBLIC UpdateResponseWithError
VAR_INPUT
	Response : I_ServerResponse;
	Message : T_MAXSTRING;
END_VAR
Response.Header.TryWriteField(HeaderKey_Status,StatusValue_Error);
Response.Header.TryWriteField(HeaderKey_Message,Message);
END_METHOD

METHOD PUBLIC UpdateResponseWithHasMoreChunks
VAR_INPUT
	Response : I_ServerResponse;
	ResponseId : T_MAXSTRING;
END_VAR
VAR
	hasMoreChunks : BOOL := TRUE;
END_VAR
Response.Header.TryWriteField(HeaderKey_ResponseId,ResponseId);
Response.Header.TryWriteField(HeaderKey_HasMoreChunks,hasMoreChunks);
END_METHOD

METHOD PUBLIC UpdateResponseWithPending
VAR_INPUT
	Response : I_ServerResponse;
	ResponseId : T_MAXSTRING;
	RetryDelayInMs : UDINT;
END_VAR
VAR
	retryDelayInMsString : T_MAXSTRING;
END_VAR
Response.Header.TryWriteField(HeaderKey_Status,StatusValue_Pending);
Response.Header.TryWriteField(HeaderKey_ResponseId, ResponseId);

IF RetryDelayInMs > 0 THEN
	retryDelayInMsString := UDINT_TO_STRING(RetryDelayInMs);
	Response.Header.TryWriteField(HeaderKey_RetryDelay, retryDelayInMsString);
END_IF
END_METHOD

METHOD PUBLIC UpdateResponseWithSessionId
VAR_INPUT
	Response : I_ServerResponse;
	SessionId : T_MAXSTRING;
END_VAR
Response.Header.TryWriteField(HeaderKey_SessionId,SessionId);
END_METHOD

METHOD PUBLIC UpdateResponseWithSuccess
VAR_INPUT
	Response : I_ServerResponse;
END_VAR
Response.Header.TryWriteField(HeaderKey_Status,StatusValue_Success);
END_METHOD

END_FUNCTION_BLOCK

// _Internal/Sessions/HeaderAccessor/I_SessionHeaderAccessor
INTERFACE I_SessionHeaderAccessor

METHOD PUBLIC TryGetSessionIdFromRequest : BOOL
VAR_INPUT
	Request : I_Request;
	Destination : REFERENCE TO T_MAXSTRING;
END_VAR
END_METHOD

METHOD PUBLIC UpdateRequestWithSessionId
VAR_INPUT
	Request : I_Request;
	SessionId : T_MAXSTRING;
END_VAR
END_METHOD

METHOD PUBLIC UpdateResponseWithSessionId
VAR_INPUT
	Response : I_ServerResponse;
	SessionId : T_MAXSTRING;
END_VAR
END_METHOD

END_INTERFACE

// _Internal/ServerResponse/HeaderAccessor/I_ServerResponseHeaderAccessor
INTERFACE I_ServerResponseHeaderAccessor

METHOD PUBLIC UpdateResponseWithAccepted
VAR_INPUT
	Response : I_ServerResponse;
END_VAR
END_METHOD

METHOD PUBLIC UpdateResponseWithBusy
VAR_INPUT
	Response : I_ServerResponse;
END_VAR
END_METHOD

METHOD PUBLIC UpdateResponseWithError
VAR_INPUT
	Response : I_ServerResponse;
	Message : T_MAXSTRING;
END_VAR
END_METHOD

METHOD PUBLIC UpdateResponseWithPending
VAR_INPUT
	Response : I_ServerResponse;
	ResponseId : T_MAXSTRING;
	RetryDelayInMs : UDINT;
END_VAR
END_METHOD

METHOD PUBLIC UpdateResponseWithSuccess
VAR_INPUT
	Response : I_ServerResponse;
END_VAR
END_METHOD

END_INTERFACE

// _Internal/ChunkedResponses/HeaderAccessor/I_ChunkedResponseHeaderAccessor
INTERFACE I_ChunkedResponseHeaderAccessor

METHOD PUBLIC TryGetResponseIdFromRequest : BOOL
VAR_INPUT
	Request : I_Request;
	Destination : ANY;
END_VAR
END_METHOD

METHOD PUBLIC TryGetSessionIdFromRequest : BOOL
VAR_INPUT
	Request : I_Request;
	Destination : REFERENCE TO T_MAXSTRING;
END_VAR
END_METHOD

METHOD PUBLIC TryGetSessionIdFromResponse : BOOL
VAR_INPUT
	Response : I_ServerResponse;
	Destination : ANY;
END_VAR
END_METHOD

METHOD PUBLIC UpdateResponseWithHasMoreChunks
VAR_INPUT
	Response : I_ServerResponse;
	ResponseId : T_MAXSTRING;
END_VAR
END_METHOD

END_INTERFACE

// _Internal/ChunkedRequests/HeaderAccessor/I_ChunkedRequestsHeaderAccessor
INTERFACE I_ChunkedRequestsHeaderAccessor

METHOD PUBLIC TryGetChunkSequenceFromRequest : BOOL
VAR_INPUT
	Request : I_Request;
	Destination : REFERENCE TO DINT;
END_VAR
END_METHOD

METHOD PUBLIC TryGetChunkTotalFromRequest : BOOL
VAR_INPUT
	Request : I_Request;
	Destination : REFERENCE TO DINT;
END_VAR
END_METHOD

METHOD PUBLIC TryGetHasMoreChunksFromRequest : BOOL
VAR_INPUT
	Request : I_Request;
	Destination : REFERENCE TO BOOL;
END_VAR
END_METHOD

METHOD PUBLIC TryGetRequestIdFromRequest : BOOL
VAR_INPUT
	Request : I_Request;
	Destination : REFERENCE TO T_MAXSTRING;
END_VAR
END_METHOD

METHOD PUBLIC TryGetSessionIdFromRequest : BOOL
VAR_INPUT
	Request : I_Request;
	Destination : REFERENCE TO T_MAXSTRING;
END_VAR
END_METHOD

END_INTERFACE

// _Internal/RPC/HeaderAccessor/I_RpcHeaderAccessor
INTERFACE I_RpcHeaderAccessor

PROPERTY PUBLIC ContentType_Json : T_MAXSTRING
GET
END_GET
END_PROPERTY

METHOD PUBLIC TryGetAcceptResponseFormatFromRequest : BOOL
VAR_INPUT
	Request : I_Request;
	Destination : ANY;
END_VAR
END_METHOD

METHOD PUBLIC TryGetContentTypeFromRequest : BOOL
VAR_INPUT
	Request : I_Request;
	Destination : ANY;
END_VAR
END_METHOD

METHOD PUBLIC TryGetMethodNameFromRequest : BOOL
VAR_INPUT
	Request : I_Request;
	Destination : ANY;
END_VAR
END_METHOD

METHOD PUBLIC TryGetTypeFromRequest : BOOL
VAR_INPUT
	Request : I_Request;
	Destination : ANY;
END_VAR
END_METHOD

END_INTERFACE

// _Internal/Sessions/Session/Session
{attribute 'linkalways'} 
{attribute 'no_explicit_call' := 'This FB is a CLASS and must be accessed using methods or properties'}
{attribute 'enable_dynamic_creation'}
FUNCTION_BLOCK Session EXTENDS Disposable IMPLEMENTS I_Session
VAR
	_id : T_MAXSTRING;
	_lastAccessedTimestamp : SystemTimestamp;
	sessionStorage : Dictionary;
END_VAR

METHOD FB_init : BOOL
VAR_INPUT
	bInitRetains : BOOL; // if TRUE, the retain variables are initialized (warm start / cold start)
	bInCopyCode : BOOL;  // if TRUE, the instance afterwards gets moved into the copy code (online change)
	SessionId : T_MAXSTRING;
END_VAR
_id := SessionId;
END_METHOD

METHOD FB_exit : BOOL
VAR_INPUT
	bInCopyCode : BOOL; // if TRUE, the exit method is called for exiting an instance that is copied afterwards (online change).
END_VAR
IF bInCopyCode THEN
	RETURN;
END_IF

DisposeAllDataFromStorage();
END_METHOD

METHOD PUBLIC AddOrUpdateStorage
VAR_INPUT
	StorageId : T_MAXSTRING;
	Source : I_SessionData;
END_VAR
sessionStorage.AddOrUpdate(StorageId, Source);
END_METHOD

METHOD PUBLIC DisposeAllDataFromStorage
VAR_INPUT
END_VAR
VAR
	enumerator : I_ForwardEnumerator;
	sessionData : I_SessionData;
END_VAR
enumerator := sessionStorage.GetEnumerator();

WHILE enumerator.MoveNext() DO
	IF enumerator.TryGet(sessionData) THEN
		sessionData.Dispose();
	END_IF
END_WHILE

enumerator.Dispose();
sessionStorage.Clear();
END_METHOD

METHOD PUBLIC DisposeDataFromStorage
VAR_INPUT
	StorageId : T_MAXSTRING;
END_VAR
VAR
	sessionData : I_SessionData;
END_VAR
IF NOT sessionStorage.TryGetValue(StorageId,sessionData) THEN
	RETURN;
END_IF

sessionData.Dispose();
sessionStorage.Remove(StorageId);
END_METHOD

PROPERTY PUBLIC Id : T_MAXSTRING
GET
Id := _id;
END_GET
END_PROPERTY

PROPERTY PUBLIC LastAccessedTimestamp : I_TimeStamp
GET
LastAccessedTimestamp := _lastAccessedTimestamp;
END_GET
END_PROPERTY

METHOD PUBLIC Refresh
VAR_INPUT
END_VAR
_lastAccessedTimestamp.SetNow();
END_METHOD

METHOD PUBLIC TryGetDataFromStorage : BOOL
VAR_INPUT
	StorageId : T_MAXSTRING;
	Destination : REFERENCE TO I_SessionData;
END_VAR
TryGetDataFromStorage := sessionStorage.TryGetValue(StorageId, Destination);
END_METHOD

END_FUNCTION_BLOCK

// _Internal/Sessions/Session/I_Session
INTERFACE I_Session Extends I_Disposable

METHOD PUBLIC AddOrUpdateStorage
VAR_INPUT
	StorageId : T_MAXSTRING;
	Source : I_SessionData;
END_VAR
END_METHOD

METHOD PUBLIC DisposeAllDataFromStorage
VAR_INPUT
END_VAR
END_METHOD

METHOD PUBLIC DisposeDataFromStorage
VAR_INPUT
	StorageId : T_MAXSTRING;
END_VAR
END_METHOD

PROPERTY PUBLIC Id : T_MAXSTRING
GET
END_GET
END_PROPERTY

PROPERTY PUBLIC LastAccessedTimestamp : I_TimeStamp
GET
END_GET
END_PROPERTY

METHOD PUBLIC Refresh
VAR_INPUT
END_VAR
END_METHOD

METHOD PUBLIC TryGetDataFromStorage : BOOL
VAR_INPUT
	StorageId : T_MAXSTRING;
	Destination : REFERENCE TO I_SessionData;
END_VAR
END_METHOD

END_INTERFACE

// _Internal/AsyncResponse/SessionData/AsyncResponseSessionData
{attribute 'linkalways'} 
{attribute 'no_explicit_call' := 'This FB is a CLASS and must be accessed using methods or properties'}
{attribute 'enable_dynamic_creation'}
FUNCTION_BLOCK AsyncResponseSessionData EXTENDS Disposable IMPLEMENTS I_AsyncResponseSessionData
VAR
	_suggestedRetryDelayInMs : UDINT;
	state : (PENDING, SUCCESS, SUCCESS_WITH_PAYLOAD, ERROR) := PENDING;
	errorMessage : T_MAXSTRING;
	pData : POINTER TO BYTE;
	dataSize : UDINT;
END_VAR

METHOD FB_init : BOOL
VAR_INPUT
	bInitRetains : BOOL; // if TRUE, the retain variables are initialized (warm start / cold start)
	bInCopyCode : BOOL;  // if TRUE, the instance afterwards gets moved into the copy code (online change)
	SuggestedRetryDelayInMs : UDINT;
END_VAR
_suggestedRetryDelayInMs := SuggestedRetryDelayInMs;
END_METHOD

METHOD FB_exit : BOOL
VAR_INPUT
	bInCopyCode : BOOL; // if TRUE, the exit method is called for exiting an instance that is copied afterwards (online change).
END_VAR
IF bInCopyCode THEN
	RETURN;
END_IF

DeletePayloadData();
END_METHOD

METHOD PUBLIC CopyPayloadData
VAR_INPUT
	PayloadDataAddress : PVOID;
	PayloadDataSize : UDINT;
END_VAR
dataSize := PayloadDataSize;
pData := __NEW(BYTE, PayloadDataSize);
memcpy(pData,PayloadDataAddress,PayloadDataSize);
END_METHOD

METHOD PRIVATE DeletePayloadData
VAR_INPUT
END_VAR
IF pData = 0 THEN
	RETURN;
END_IF

__DELETE(pData);
dataSize := 0;
END_METHOD

METHOD PUBLIC Error
VAR_INPUT
	Message : T_MAXSTRING;
END_VAR
IF state <> PENDING THEN
	RETURN;
END_IF

state := ERROR;
errorMessage := Message;
END_METHOD

PROPERTY PUBLIC IsPending : BOOL
GET
IsPending := state = PENDING;
END_GET
END_PROPERTY

METHOD PUBLIC Success
VAR_INPUT
END_VAR
IF state <> PENDING THEN
	RETURN;
END_IF

state := SUCCESS;
END_METHOD

METHOD PUBLIC SuccessWithPayload
VAR_INPUT
	PayloadDataAddress : PVOID;
	PayloadDataSize : UDINT;
END_VAR
IF state <> PENDING THEN
	RETURN;
END_IF

state := SUCCESS_WITH_PAYLOAD;
CopyPayloadData(PayloadDataAddress, PayloadDataSize);
END_METHOD

PROPERTY PUBLIC SuggestedRetryDelayInMs : UDINT
GET
SuggestedRetryDelayInMs := _suggestedRetryDelayInMs;
END_GET
SET
PUBLIC 
VAR
END_VAR
_suggestedRetryDelayInMs := SuggestedRetryDelayInMs;
END_SET
END_PROPERTY

METHOD PUBLIC TryUpdateServerResponse : BOOL
VAR_INPUT
	Response : I_ServerResponse;
END_VAR
IF State = SUCCESS_WITH_PAYLOAD THEN
	Response.SuccessWithPayload(pData,dataSize);
	TryUpdateServerResponse := TRUE;
	RETURN;
END_IF

IF State = SUCCESS THEN
	Response.Success();
	TryUpdateServerResponse := TRUE;
	RETURN;
END_IF

IF state = ERROR THEN
	Response.Error(errorMessage);
	TryUpdateServerResponse := TRUE;
	RETURN;
END_IF
END_METHOD

END_FUNCTION_BLOCK

// _Internal/AsyncResponse/Proxy/AsyncResponseSessionDataProxy
{attribute 'linkalways'} 
{attribute 'no_explicit_call' := 'This FB is a CLASS and must be accessed using methods or properties'}
{attribute 'enable_dynamic_creation'}
FUNCTION_BLOCK AsyncResponseSessionDataProxy EXTENDS Disposable IMPLEMENTS I_AsyncResponseSessionData
VAR
	sessionStorage : I_SessionStorage;
	sessionId : T_MAXSTRING;
	responseId : T_MAXSTRING;
END_VAR

METHOD FB_init : BOOL
VAR_INPUT
	bInitRetains : BOOL; // if TRUE, the retain variables are initialized (warm start / cold start)
	bInCopyCode : BOOL;  // if TRUE, the instance afterwards gets moved into the copy code (online change)
	SessionStorage : I_SessionStorage;
	SessionId : T_MAXSTRING;
	ResponseId : T_MAXSTRING;
END_VAR
THIS^.sessionStorage := SessionStorage;
THIS^.sessionId := SessionId;
THIS^.responseId := ResponseId;
END_METHOD

METHOD PROTECTED TryGetAsyncResponseSessionData : BOOL;
VAR_INPUT
	Destination : REFERENCE TO I_AsyncResponseSessionData;
END_VAR
VAR
	sessionData : I_SessionData;
	asyncSessionData : I_AsyncResponseSessionData;
END_VAR
IF NOT sessionStorage.TryRetreiveSessionDataById(sessionId, responseId, sessionData) THEN
	RETURN;
END_IF

IF NOT __QUERYINTERFACE(sessionData, asyncSessionData) THEN
	RETURN;
END_IF

Destination := asyncSessionData;
TryGetAsyncResponseSessionData := TRUE;
END_METHOD

METHOD PUBLIC Error
VAR_INPUT
	Message : T_MAXSTRING;
END_VAR
VAR
	asyncReponseSessionData : I_AsyncResponseSessionData;
END_VAR
IF NOT TryGetAsyncResponseSessionData(asyncReponseSessionData) THEN
	RETURN;
END_IF

asyncReponseSessionData.Error(Message);
END_METHOD

PROPERTY PUBLIC IsPending : BOOL
GET
VAR
	asyncReponseSessionData : I_AsyncResponseSessionData;
END_VAR
IF NOT TryGetAsyncResponseSessionData(asyncReponseSessionData) THEN
	RETURN;
END_IF

IsPending := asyncReponseSessionData.IsPending;
END_GET
END_PROPERTY

METHOD PUBLIC Success
VAR_INPUT
END_VAR
VAR
	asyncReponseSessionData : I_AsyncResponseSessionData;
END_VAR
IF NOT TryGetAsyncResponseSessionData(asyncReponseSessionData) THEN
	RETURN;
END_IF

asyncReponseSessionData.Success();
END_METHOD

METHOD PUBLIC SuccessWithPayload
VAR_INPUT
	PayloadDataAddress : PVOID;
	PayloadDataSize : UDINT;
END_VAR
VAR
	asyncReponseSessionData : I_AsyncResponseSessionData;
END_VAR
IF NOT TryGetAsyncResponseSessionData(asyncReponseSessionData) THEN
	RETURN;
END_IF

asyncReponseSessionData.SuccessWithPayload(PayloadDataAddress, PayloadDataSize);
END_METHOD

PROPERTY PUBLIC SuggestedRetryDelayInMs : UDINT
GET
VAR
	asyncReponseSessionData : I_AsyncResponseSessionData;
END_VAR
IF NOT TryGetAsyncResponseSessionData(asyncReponseSessionData) THEN
	RETURN;
END_IF

SuggestedRetryDelayInMs := asyncReponseSessionData.SuggestedRetryDelayInMs;
END_GET
SET
PUBLIC 
VAR
	asyncReponseSessionData : I_AsyncResponseSessionData;
END_VAR
IF NOT TryGetAsyncResponseSessionData(asyncReponseSessionData) THEN
	RETURN;
END_IF

asyncReponseSessionData.SuggestedRetryDelayInMs := SuggestedRetryDelayInMs;
END_SET
END_PROPERTY

METHOD PUBLIC TryUpdateServerResponse : BOOL
VAR_INPUT
	Response : I_ServerResponse;
END_VAR
VAR
	asyncReponseSessionData : I_AsyncResponseSessionData;
END_VAR
IF NOT TryGetAsyncResponseSessionData(asyncReponseSessionData) THEN
	RETURN;
END_IF

TryUpdateServerResponse := asyncReponseSessionData.TryUpdateServerResponse(Response);
END_METHOD

END_FUNCTION_BLOCK

// _Internal/AsyncResponse/Middleware/AsyncResponseMiddleware
FUNCTION_BLOCK AsyncResponseMiddleware EXTENDS MiddlewareBase
VAR
	asyncResponseManager : I_AsyncResponseManager;
END_VAR

METHOD FB_init : BOOL
VAR_INPUT
	bInitRetains : BOOL; // if TRUE, the retain variables are initialized (warm start / cold start)
	bInCopyCode : BOOL;  // if TRUE, the instance afterwards gets moved into the copy code (online change)
	AsyncResponseManager : I_AsyncResponseManager;
END_VAR
This^.asyncResponseManager := AsyncResponseManager;
END_METHOD

METHOD PUBLIC Handle
VAR_INPUT
	Request : I_Request;
	Response : I_ServerResponse;
END_VAR
IF asyncResponseManager.TryHandleIncomingRequest(Request, Response) THEN
	RETURN;
END_IF

Next(Request, Response);
END_METHOD

END_FUNCTION_BLOCK

// _Internal/Middleware/Base/MiddlewareBase
{attribute 'linkalways'} 
{attribute 'no_explicit_call' := 'This FB is a CLASS and must be accessed using methods or properties'}
{attribute 'enable_dynamic_creation'}
FUNCTION_BLOCK ABSTRACT MiddlewareBase implements I_Middleware
VAR
	_next : I_Middleware;
END_VAR

METHOD PROTECTED Next
VAR_INPUT
	Request : I_Request;
	Response : I_ServerResponse;
END_VAR
IF _next = 0 THEN
	RETURN;
END_IF

_next.Handle(Request, Response);
END_METHOD

METHOD PUBLIC ABSTRACT Handle
VAR_INPUT
	Request : I_Request;
	Response : I_ServerResponse;
END_VAR
// Call next to pass the request and response to the next handler
// Next(Request, Response);
END_METHOD

PROPERTY PUBLIC NextMiddleware : I_Middleware
GET
NextMiddleware := _next;
END_GET
SET
_next := NextMiddleware;
END_SET
END_PROPERTY

END_FUNCTION_BLOCK

// _Internal/Middleware/Interface/I_Middleware
INTERFACE I_Middleware

METHOD Handle
VAR_INPUT
	Request : I_Request;
	Response : I_ServerResponse;
END_VAR
END_METHOD

PROPERTY PUBLIC NextMiddleware : I_Middleware
GET
END_GET
SET
END_SET
END_PROPERTY

END_INTERFACE

// _Internal/ChunkedRequests/ChunkedRequest/ChunkedRequest
{attribute 'linkalways'} 
{attribute 'no_explicit_call' := 'This FB is a CLASS and must be accessed using methods or properties'}
{attribute 'enable_dynamic_creation'}
FUNCTION_BLOCK ChunkedRequest EXTENDS Disposable IMPLEMENTS I_Request
VAR
	request : I_Request;
	chunkedRequestData : REFERENCE TO I_ChunkedRequestData;
END_VAR

METHOD FB_init : BOOL
VAR_INPUT
	bInitRetains : BOOL; // if TRUE, the retain variables are initialized (warm start / cold start)
	bInCopyCode : BOOL;  // if TRUE, the instance afterwards gets moved into the copy code (online change)
	Request : I_Request;
	ChunkedRequestData : Reference to I_ChunkedRequestData;
END_VAR
THIS^.request := Request;
this^.chunkedRequestData ref= ChunkedRequestData;
END_METHOD

PROPERTY PUBLIC CreatedTimestamp : I_Timestamp
GET
CreatedTimestamp := request.CreatedTimestamp;
END_GET
END_PROPERTY

PROPERTY PUBLIC Header : I_Header
GET
Header := request.Header;
END_GET
END_PROPERTY

PROPERTY PUBLIC PayloadAddress : POINTER TO STRING
GET
IF chunkedRequestData = 0 THEN
	RETURN;
END_IF

PayloadAddress := chunkedRequestData.PayloadAddress;
END_GET
END_PROPERTY

PROPERTY PUBLIC PayloadSizeInBytes : UDINT
GET
IF chunkedRequestData = 0 THEN
	RETURN;
END_IF

PayloadSizeInBytes := chunkedRequestData.PayloadSizeInBytes;
END_GET
END_PROPERTY

END_FUNCTION_BLOCK

// _Internal/ChunkedRequests/SessionData/ChunkedRequestData
{attribute 'linkalways'} 
{attribute 'no_explicit_call' := 'This FB is a CLASS and must be accessed using methods or properties'}
{attribute 'enable_dynamic_creation'}
FUNCTION_BLOCK ChunkedRequestData EXTENDS Disposable IMPLEMENTS I_ChunkedRequestData
VAR
	maximumChunkSizeInBytes : UDINT;
	totalReceivedChunks : UDINT;
	totalExpectedChunks : UDINT;
	pPayloadBuffer : POINTER TO STRING;
	payloadBufferSize : UDINT;
END_VAR

METHOD FB_init : BOOL
VAR_INPUT
	bInitRetains : BOOL; // if TRUE, the retain variables are initialized (warm start / cold start)
	bInCopyCode : BOOL;  // if TRUE, the instance afterwards gets moved into the copy code (online change)
	ChunkSizeInBytes : UDINT;
	ChunkCount : UDINT;
END_VAR
maximumChunkSizeInBytes := ChunkSizeInBytes;
totalExpectedChunks := ChunkCount;
CreateBuffer(ChunkSizeInBytes * ChunkCount);
END_METHOD

METHOD FB_exit : BOOL
VAR_INPUT
	bInCopyCode : BOOL; // if TRUE, the exit method is called for exiting an instance that is copied afterwards (online change).
END_VAR
IF bInCopyCode THEN
	RETURN;
END_IF

DestroyBuffer();
END_METHOD

METHOD PRIVATE CreateBuffer
VAR_INPUT
	SizeInBytes : UDINT;
END_VAR
payloadBufferSize := SizeInBytes;
pPayloadBuffer := __NEW(BYTE, SizeInBytes);
memset(pPayloadBuffer, 0, SizeInBytes);
END_METHOD

METHOD PRIVATE DestroyBuffer
VAR_INPUT
END_VAR
IF pPayloadBuffer = 0 THEN
	RETURN;
END_IF

__DELETE(pPayloadBuffer);
pPayloadBuffer := 0;
END_METHOD

PROPERTY PUBLIC IsComplete : BOOL
GET
IsComplete := totalReceivedChunks = totalExpectedChunks;
END_GET
END_PROPERTY

PROPERTY PUBLIC PayloadAddress : POINTER TO STRING
GET
PayloadAddress := pPayloadBuffer;
END_GET
END_PROPERTY

PROPERTY PUBLIC PayloadSizeInBytes : UDINT
GET
PayloadSizeInBytes := payloadBufferSize;
END_GET
END_PROPERTY

METHOD PUBLIC TryAddChunkedPayload : BOOL;
VAR_INPUT
	PayloadAddress : POINTER TO STRING;
	PayloadSize : DINT;
	ChunkSequence : DINT;
END_VAR
VAR
	offset : UDINT;
	pBufferChunkLocation : POINTER TO BYTE;
END_VAR
IF totalReceivedChunks >= totalExpectedChunks THEN
	RETURN;
END_IF

IF DINT_TO_UDINT(PayloadSize) > maximumChunkSizeInBytes THEN
	RETURN;
END_IF

IF ChunkSequence <= 0 THEN
	RETURN;
END_IF

concat2(pPayloadBuffer, PayloadAddress, pPayloadBuffer, payloadBufferSize);
totalReceivedChunks := totalReceivedChunks + 1;

TryAddChunkedPayload := TRUE;
END_METHOD

END_FUNCTION_BLOCK

// _Internal/ChunkedRequests/SessionData/I_ChunkedRequestData
INTERFACE I_ChunkedRequestData EXTENDS I_SessionData

PROPERTY PUBLIC IsComplete : BOOL
GET
END_GET
END_PROPERTY

PROPERTY PUBLIC PayloadAddress : POINTER TO STRING
GET
END_GET
END_PROPERTY

PROPERTY PUBLIC PayloadSizeInBytes : UDINT
GET
END_GET
END_PROPERTY

METHOD PUBLIC TryAddChunkedPayload : BOOL;
VAR_INPUT
	PayloadAddress : POINTER TO STRING;
	PayloadSize : DINT;
	ChunkSequence : DINT;
END_VAR
END_METHOD

END_INTERFACE

// _Internal/ChunkedRequests/Manager/ChunkedRequestsManager
{attribute 'linkalways'} 
{attribute 'no_explicit_call' := 'This FB is a CLASS and must be accessed using methods or properties'}
{attribute 'enable_dynamic_creation'}
FUNCTION_BLOCK ChunkedRequestsManager IMPLEMENTS I_ChunkedRequestsManager
VAR
	maximumChunkSizeInBytes : UDINT;
	sessionStorage : I_SessionStorage;
	headerAccessor : I_ChunkedRequestsHeaderAccessor;
END_VAR

METHOD FB_init : BOOL
VAR_INPUT
	bInitRetains : BOOL; // if TRUE, the retain variables are initialized (warm start / cold start)
	bInCopyCode : BOOL;  // if TRUE, the instance afterwards gets moved into the copy code (online change)
	MaximumChunkSizeInBytes : UDINT;
	SessionStorage : I_SessionStorage;
	HeaderAccessor : I_ChunkedRequestsHeaderAccessor;
END_VAR
THIS^.maximumChunkSizeInBytes := MaximumChunkSizeInBytes;
THIS^.sessionStorage := SessionStorage;
THIS^.headerAccessor := HeaderAccessor;
END_METHOD

METHOD PRIVATE CreateChunkedRequestData : I_ChunkedRequestData
VAR_INPUT
	RequestChunkSizeInBytes : UDINT;
	RequestChunkCount : UDINT;
END_VAR
VAR
	pChunkedRequestData : POINTER TO ChunkedRequestData;
END_VAR
pChunkedRequestData := __NEW(ChunkedRequestData(ChunkSizeInBytes := RequestChunkSizeInBytes, ChunkCount := RequestChunkCount));
CreateChunkedRequestData := pChunkedRequestData^;
END_METHOD

METHOD PUBLIC TryHandleIncomingRequest : BOOL
VAR_INPUT
	Request : I_Request;
	Response : I_ServerResponse;
	NextMidleware : I_Middleware;
END_VAR
VAR 
	hasChunkSequenceHeader : BOOL;
	chunkSequence : DINT;
	hasChunkTotalHeader : BOOL;
	chunkTotal : DINT;
	hasMoreChunksHeader : BOOL;
	hasMoreChunks : BOOL;
	requestId : T_MAXSTRING;
	sessionId : T_MAXSTRING;
	sessionData : I_SessionData;
	chunkedRequestData : I_ChunkedRequestData;
	chunkedRequest : ChunkedRequest(Request, chunkedRequestData);
END_VAR
hasChunkSequenceHeader := headerAccessor.TryGetChunkSequenceFromRequest(Request, chunkSequence);
hasChunkTotalHeader := headerAccessor.TryGetChunkTotalFromRequest(Request, chunkTotal);
hasMoreChunksHeader := headerAccessor.TryGetHasMoreChunksFromRequest(Request, hasMoreChunks);

IF (NOT hasChunkSequenceHeader) AND (NOT hasChunkTotalHeader) AND (NOT hasMoreChunksHeader) THEN
	// this is not a chunked request, simply return and it will be handled by the next middleware automatically.
	RETURN;
END_IF

// when reaching here we know that the request has at least one of the headers associated with chunked requests
// from this point on, we simply validate until we know we have all the required parts. 

IF NOT hasChunkSequenceHeader THEN
	response.Error('Chunked Request found, but chunk sequence header data is missing');
	TryHandleIncomingRequest := TRUE;
	RETURN;
END_IF

IF chunkSequence = 0 THEN
	response.Error('Chunk sequence 0 received, chunks must start from 1');
	TryHandleIncomingRequest := TRUE;
	RETURN;
END_IF

IF NOT hasChunkTotalHeader THEN
	response.Error('Chunked Request found, but chunk total header data is missing');
	TryHandleIncomingRequest := TRUE;
	RETURN;
END_IF

IF chunkSequence > chunkTotal THEN
	response.Error('Chunk sequence is greater than the chunk total');
	TryHandleIncomingRequest := TRUE;
	RETURN;
END_IF

IF NOT hasMoreChunksHeader THEN
	response.Error('Chunked Request found, but has more chunks header data is missing');
	TryHandleIncomingRequest := TRUE;
	RETURN;
END_IF

IF NOT headerAccessor.TryGetRequestIdFromRequest(Request, requestId) THEN
	response.Error('Chunked Request found, but request id header data is missing');
	TryHandleIncomingRequest := TRUE;
	RETURN;
END_IF

IF NOT headerAccessor.TryGetSessionIdFromRequest(Request, sessionId) THEN
	response.Error('Chunked Request found, but session id header data is missing');
	TryHandleIncomingRequest := TRUE;
	RETURN;
END_IF

// at this point we know we have all of the data required for handling a chunked request

IF NOT sessionStorage.TryRetreiveSessionDataById(sessionId, requestId, sessionData) THEN	
	chunkedRequestData := CreateChunkedRequestData(maximumChunkSizeInBytes, DINT_TO_UDINT(chunkTotal));
	sessionStorage.TryStoreSessionDataById(sessionId, requestId, chunkedRequestData);
ELSIF NOT __QUERYINTERFACE(sessionData, chunkedRequestData) THEN
	response.Error('Server was unable to retreive previous session data as chunked request data');
	TryHandleIncomingRequest := TRUE;
	RETURN;
END_IF

IF NOT chunkedRequestData.TryAddChunkedPayload(request.PayloadAddress, request.PayloadSizeInBytes, chunkSequence) THEN
	response.Error('Unable to store request payload in chunk session storage');
	sessionStorage.DisposeSessionDataById(sessionId, requestId);
	TryHandleIncomingRequest := TRUE;
	RETURN;
END_IF

IF NOT chunkedRequestData.IsComplete THEN
	Response.Accepted();
	TryHandleIncomingRequest := TRUE;
	RETURN;
END_IF

NextMidleware.Handle(chunkedRequest, Response);
sessionStorage.DisposeSessionDataById(sessionId, requestId);
TryHandleIncomingRequest := TRUE;
END_METHOD

END_FUNCTION_BLOCK

// _Internal/ChunkedRequests/Manager/I_ChunkedRequestsManager
INTERFACE I_ChunkedRequestsManager

METHOD PUBLIC TryHandleIncomingRequest : BOOL
VAR_INPUT
	Request : I_Request;
	Response : I_ServerResponse;
	NextMidleware : I_Middleware;
END_VAR
END_METHOD

END_INTERFACE

// _Internal/ChunkedRequests/Middleware/ChunkedRequestsMiddleware
{attribute 'linkalways'} 
{attribute 'no_explicit_call' := 'This FB is a CLASS and must be accessed using methods or properties'}
{attribute 'enable_dynamic_creation'}
FUNCTION_BLOCK ChunkedRequestsMiddleware EXTENDS MiddlewareBase
VAR
	chunkedRequestsManager : I_ChunkedRequestsManager;
END_VAR

METHOD FB_init : BOOL
VAR_INPUT
	bInitRetains : BOOL; // if TRUE, the retain variables are initialized (warm start / cold start)
	bInCopyCode : BOOL;  // if TRUE, the instance afterwards gets moved into the copy code (online change)
	ChunkedRequestsManager : I_ChunkedRequestsManager;
END_VAR
THIS^.chunkedRequestsManager := ChunkedRequestsManager;
END_METHOD

METHOD PUBLIC Handle
VAR_INPUT
	Request : I_Request;
	Response : I_ServerResponse;
END_VAR
VAR
	hasMoreChunks : BOOL;
END_VAR
IF chunkedRequestsManager.TryHandleIncomingRequest(Request, Response, NextMiddleware) THEN
	RETURN;
END_IF

Next(Request, Response);
END_METHOD

END_FUNCTION_BLOCK

// _Internal/ChunkedResponses/Manager/ChunkedResponseManager
{attribute 'linkalways'} 
{attribute 'no_explicit_call' := 'This FB is a CLASS and must be accessed using methods or properties'}
{attribute 'enable_dynamic_creation'}
FUNCTION_BLOCK ChunkedResponseManager IMPLEMENTS I_ChunkedResponseManager
VAR
	maximumChunkSizeInBytes : UDINT;
	sessionStorage : I_SessionStorage;
	responseIdGenerator : I_ResponseIdGenerator;
	headerAccessor : I_ChunkedResponseHeaderAccessor;
END_VAR

METHOD FB_init : BOOL
VAR_INPUT
	bInitRetains : BOOL; // if TRUE, the retain variables are initialized (warm start / cold start)
	bInCopyCode : BOOL;  // if TRUE, the instance afterwards gets moved into the copy code (online change)
	MaximumChunkSizeInBytes : UDINT;
	SessionStorage : I_SessionStorage;
	ResponseIdGenerator : I_ResponseIdGenerator;
	HeaderAccessor : I_ChunkedResponseHeaderAccessor;
END_VAR
THIS^.maximumChunkSizeInBytes := MaximumChunkSizeInBytes;
THIS^.sessionStorage := SessionStorage;
THIS^.responseIdGenerator := ResponseIdGenerator;
This^.headerAccessor := HeaderAccessor;
END_METHOD

METHOD PUBLIC CreateChunkedResponseData : I_ChunkedResponseData
VAR_INPUT
	DataAddress : PVOID;
	DataSize : UDINT;
END_VAR
VAR
	pChunkedResponseData : POINTER TO ChunkedResponseData;
END_VAR
pChunkedResponseData := __NEW(ChunkedResponseData(Address := DataAddress, Size:=DataSize));
CreateChunkedResponseData := pChunkedResponseData^;
END_METHOD

METHOD PUBLIC HandleSuccessWithPayload
VAR_INPUT
	OriginalResponse : I_ServerResponse;
	SourceAddress : PVOID;
	SourceSize : UDINT;
END_VAR
VAR
	sessionId : T_MAXSTRING;
	responseId : T_MAXSTRING;
	chunkedResponseData : I_ChunkedResponseData;
END_VAR
IF SourceSize <= maximumChunkSizeInBytes THEN
	OriginalResponse.SuccessWithPayload(SourceAddress, SourceSize);
	RETURN;
END_IF

IF NOT headerAccessor.TryGetSessionIdFromResponse(OriginalResponse,sessionId) THEN
	OriginalResponse.Error('Unable to chunk oversized response without a sessionId');
	RETURN;
END_IF

chunkedResponseData := CreateChunkedResponseData(SourceAddress, SourceSize);
responseId := responseIdGenerator.Generate();

IF NOT sessionStorage.TryStoreSessionDataById(sessionId, responseId, chunkedResponseData) THEN
	OriginalResponse.Error('Unable to store oversized response');
	chunkedResponseData.Dispose();
	RETURN;
END_IF

headerAccessor.UpdateResponseWithHasMoreChunks(OriginalResponse, responseId);
chunkedResponseData.SendNextChunk(OriginalResponse, maximumChunkSizeInBytes);
END_METHOD

METHOD PUBLIC TryHandleIncomingRequest : BOOL
VAR_INPUT
	Request : I_Request;
	Response : I_ServerResponse;
END_VAR
VAR
	responseId : T_MAXSTRING;
	sessionId : T_MAXSTRING;
	sessionData : I_SessionData;
	chunkedResponseData : I_ChunkedResponseData;
END_VAR
IF NOT headerAccessor.TryGetResponseIdFromRequest(Request, responseId) THEN
	RETURN;
END_IF

IF NOT headerAccessor.TryGetSessionIdFromRequest(Request, sessionId) THEN
	RETURN;
END_IF

IF NOT sessionStorage.TryRetreiveSessionDataById(sessionId, responseId, sessionData) THEN
	RETURN;
END_IF

IF NOT __QUERYINTERFACE(sessionData, chunkedResponseData) THEN
	RETURN;
END_IF

IF chunkedResponseData.SizeRemaining > maximumChunkSizeInBytes THEN
	headerAccessor.UpdateResponseWithHasMoreChunks(Response, responseId);
END_IF

chunkedResponseData.SendNextChunk(Response, maximumChunkSizeInBytes);

IF chunkedResponseData.SendComplete THEN
	sessionStorage.DisposeSessionDataById(sessionId, responseId);
END_IF

TryHandleIncomingRequest := TRUE;
END_METHOD

END_FUNCTION_BLOCK

// _Internal/ChunkedResponses/Manager/I_ChunkedResponseManager
INTERFACE I_ChunkedResponseManager

METHOD PUBLIC HandleSuccessWithPayload;
VAR_INPUT
	OriginalResponse : I_ServerResponse;
	SourceAddress : PVOID;
	SourceSize : UDINT;
END_VAR
END_METHOD

METHOD PUBLIC TryHandleIncomingRequest : BOOL
VAR_INPUT
	Request : I_Request;
	Response : I_ServerResponse;
END_VAR
END_METHOD

END_INTERFACE

// _Internal/ChunkedResponses/SessionData/ChunkedResponseData
{attribute 'linkalways'} 
{attribute 'no_explicit_call' := 'This FB is a CLASS and must be accessed using methods or properties'}
{attribute 'enable_dynamic_creation'}
FUNCTION_BLOCK ChunkedResponseData EXTENDS Disposable IMPLEMENTS I_ChunkedResponseData
VAR
	pData : POINTER TO BYTE;
	size : UDINT;
	currentPointerLocation : PVOID;
	remainingLengthToSendInBytes : UDINT;
END_VAR

METHOD FB_init : BOOL
VAR_INPUT
	bInitRetains : BOOL; // if TRUE, the retain variables are initialized (warm start / cold start)
	bInCopyCode : BOOL;  // if TRUE, the instance afterwards gets moved into the copy code (online change)
	Address : PVOID;
	Size : UDINT;
END_VAR
StoreData(Address, Size);
END_METHOD

METHOD FB_exit : BOOL
VAR_INPUT
	bInCopyCode : BOOL; // if TRUE, the exit method is called for exiting an instance that is copied afterwards (online change).
END_VAR
IF bInCopyCode THEN
	RETURN;
END_IF

IF pData <> 0 THEN
	__DELETE(pData);
END_IF
END_METHOD

METHOD PRIVATE StoreData
VAR_INPUT
	Address : PVOID;
	Size : UDINT;
END_VAR
pData := __NEW(BYTE, Size);
THIS^.size := Size;
memcpy(pData, Address, Size);
currentPointerLocation := pData;
remainingLengthToSendInBytes := Size;
END_METHOD

PROPERTY PUBLIC SendComplete : BOOL
GET
SendComplete := remainingLengthToSendInBytes = 0;
END_GET
END_PROPERTY

METHOD PUBLIC SendNextChunk
VAR_INPUT
	Response : I_ServerResponse;
	Size : UDINT;
END_VAR
VAR
	sendSize : UDINT;
END_VAR
IF SendComplete THEN 
	Response.Error('No further data to send');
	RETURN;
END_IF

sendSize := Size - 1;

IF Size > remainingLengthToSendInBytes THEN 
	sendSize := remainingLengthToSendInBytes;
END_IF

Response.SuccessWithPayload(currentPointerLocation, sendSize);

currentPointerLocation := currentPointerLocation + sendSize;
remainingLengthToSendInBytes := remainingLengthToSendInBytes - sendSize;
END_METHOD

PROPERTY SizeRemaining : UDINT
GET
SizeRemaining := remainingLengthToSendInBytes;
END_GET
END_PROPERTY

END_FUNCTION_BLOCK

// _Internal/ChunkedResponses/SessionData/I_ChunkedResponseData
INTERFACE I_ChunkedResponseData EXTENDS I_SessionData

PROPERTY PUBLIC SendComplete : BOOL
GET
END_GET
END_PROPERTY

METHOD PUBLIC SendNextChunk
VAR_INPUT
	Response : I_ServerResponse;
	Size : UDINT;
END_VAR
END_METHOD

PROPERTY SizeRemaining : UDINT
GET
END_GET
END_PROPERTY

END_INTERFACE

// _Internal/ChunkedResponses/Middleware/ChunkedResponsesMiddleware
{attribute 'linkalways'} 
{attribute 'no_explicit_call' := 'This FB is a CLASS and must be accessed using methods or properties'}
{attribute 'enable_dynamic_creation'}
FUNCTION_BLOCK ChunkedResponsesMiddleware EXTENDS MiddlewareBase
VAR
	chunkedResponseManager : I_ChunkedResponseManager;
END_VAR

METHOD FB_init : BOOL
VAR_INPUT
	bInitRetains : BOOL; // if TRUE, the retain variables are initialized (warm start / cold start)
	bInCopyCode : BOOL;  // if TRUE, the instance afterwards gets moved into the copy code (online change)
	ChunkedResponseManager : I_ChunkedResponseManager;
END_VAR
THIS^.chunkedResponseManager := ChunkedResponseManager;
END_METHOD

METHOD PUBLIC Handle
VAR_INPUT
	Request : I_Request;
	Response : I_ServerResponse;
END_VAR
VAR
	chunkableServerResponse : ChunkableServerResponse(Response, chunkedResponseManager);
END_VAR
IF chunkedResponseManager.TryHandleIncomingRequest(Request, Response) THEN
	RETURN;
END_IF

Next(Request, chunkableServerResponse);
END_METHOD

END_FUNCTION_BLOCK

// _Internal/ChunkedResponses/ServerResponse/ChunkableServerResponse
{attribute 'linkalways'} 
{attribute 'no_explicit_call' := 'This FB is a CLASS and must be accessed using methods or properties'}
{attribute 'enable_dynamic_creation'}
FUNCTION_BLOCK ChunkableServerResponse IMPLEMENTS I_ServerResponse
VAR
	serverResponse : I_ServerResponse;
	chunkedResponseManager : I_ChunkedResponseManager;
END_VAR

METHOD FB_init : BOOL
VAR_INPUT
	bInitRetains : BOOL; // if TRUE, the retain variables are initialized (warm start / cold start)
	bInCopyCode : BOOL;  // if TRUE, the instance afterwards gets moved into the copy code (online change)
	ServerResponse : I_ServerResponse;
	ChunkedResponseManager : I_ChunkedResponseManager;
END_VAR
THIS^.serverResponse := ServerResponse;
This^.chunkedResponseManager := ChunkedResponseManager;
END_METHOD

METHOD PUBLIC Accepted
VAR_INPUT
END_VAR
serverResponse.Accepted();
END_METHOD

METHOD PUBLIC Busy
VAR_INPUT
END_VAR
serverResponse.Busy();
END_METHOD

METHOD PUBLIC Error
VAR_INPUT
	Message : T_MAXSTRING;
END_VAR
serverResponse.Error(Message);
END_METHOD

PROPERTY PUBLIC Header : I_Header
GET
Header := serverResponse.Header;
END_GET
END_PROPERTY

PROPERTY PUBLIC HeadersSent : BOOL
GET
HeadersSent := serverResponse.HeadersSent;
END_GET
END_PROPERTY

METHOD PUBLIC Pending
VAR_INPUT
	ResponseId : REFERENCE TO T_MAXSTRING;
	RetryDelayInMs : UDINT;
END_VAR
serverResponse.Pending(ResponseId, RetryDelayInMs);
END_METHOD

METHOD PUBLIC Success
VAR_INPUT
END_VAR
serverResponse.Success();
END_METHOD

METHOD PUBLIC SuccessWithPayload
VAR_INPUT
	PayloadDataAddress : PVOID;
	PayloadDataSize : UDINT;
END_VAR
chunkedResponseManager.HandleSuccessWithPayload(serverResponse, PayloadDataAddress, PayloadDataSize);
END_METHOD

END_FUNCTION_BLOCK

// _Internal/ServerResponse/ServerResponse
{attribute 'linkalways'} 
{attribute 'no_explicit_call' := 'This FB is a CLASS and must be accessed using methods or properties'}
{attribute 'enable_dynamic_creation'}
FUNCTION_BLOCK ServerResponse IMPLEMENTS I_ServerResponse
VAR
	_header : Header(0);
	_sent : BOOL := FALSE;
	responseData : ResponseData;
	headerAccessor : I_ServerResponseHeaderAccessor;
END_VAR

METHOD FB_init : BOOL
VAR_INPUT
	bInitRetains : BOOL; // if TRUE, the retain variables are initialized (warm start / cold start)
	bInCopyCode : BOOL;  // if TRUE, the instance afterwards gets moved into the copy code (online change)
	HeaderAccessor : I_ServerResponseHeaderAccessor;
END_VAR
THIS^.headerAccessor := HeaderAccessor;
memset(ADR(responseData),0,SIZEOF(responseData));
END_METHOD

METHOD PRIVATE CompleteResponseWithoutPayload
VAR_INPUT
END_VAR
_sent := TRUE;
_header.ToString(responseData.Header);
memset(ADR(responseData.Payload),0,SIZEOF(responseData.Payload));
END_METHOD

METHOD PRIVATE CompleteResponseWithPayload
VAR_INPUT
	PayloadDataAddress : PVOID;
	PayloadDataSize : UDINT;
END_VAR
_sent := TRUE;
_header.ToString(responseData.Header);
memcpy(ADR(responseData.Payload),PayloadDataAddress,PayloadDataSize);
END_METHOD

METHOD PUBLIC Accepted
VAR_INPUT
END_VAR
IF _sent THEN
	RETURN;
END_IF

headerAccessor.UpdateResponseWithAccepted(THIS^);
CompleteResponseWithoutPayload();
END_METHOD

METHOD PUBLIC Busy
VAR_INPUT
END_VAR
IF _sent THEN
	RETURN;
END_IF

headerAccessor.UpdateResponseWithBusy(THIS^);
CompleteResponseWithoutPayload();
END_METHOD

METHOD PUBLIC Error
VAR_INPUT
	Message : T_MAXSTRING;
END_VAR
IF _sent THEN
	RETURN;
END_IF

headerAccessor.UpdateResponseWithError(THIS^, Message);
CompleteResponseWithoutPayload();
END_METHOD

PROPERTY PUBLIC Header : I_Header
GET
Header := _header;
END_GET
END_PROPERTY

PROPERTY PUBLIC HeadersSent : BOOL
GET
HeadersSent := _sent;
END_GET
END_PROPERTY

METHOD PUBLIC Pending
VAR_INPUT
	ResponseId : REFERENCE TO T_MAXSTRING;
	RetryDelayInMs : UDINT;
END_VAR
IF _sent THEN
	RETURN;
END_IF

IF (NOT __ISVALIDREF(ResponseId)) OR_ELSE ResponseId = '' THEN
	Error('Unable to mark response as pending without ResponseId');
	RETURN;
END_IF

headerAccessor.UpdateResponseWithPending(THIS^, ResponseId, RetryDelayInMs);
CompleteResponseWithoutPayload();
END_METHOD

METHOD PUBLIC Success
VAR_INPUT
END_VAR
VAR
	errorMessage : T_MAXSTRING;
END_VAR
IF _sent THEN
	RETURN;
END_IF

headerAccessor.UpdateResponseWithSuccess(THIS^);
CompleteResponseWithoutPayload();
END_METHOD

METHOD PUBLIC SuccessWithPayload
VAR_INPUT
	PayloadDataAddress : PVOID;
	PayloadDataSize : UDINT;
END_VAR
VAR
	errorMessage : T_MAXSTRING;
END_VAR
IF _sent THEN
	RETURN;
END_IF

IF PayloadDataSize > SIZEOF(responseData.Payload) THEN
	errorMessage := 'Payload too big to transmit. Maximum : ';
	errorMessage := concat(errorMessage, UDINT_TO_STRING(SIZEOF(responseData.Payload)));
	errorMessage := concat(errorMessage, ', Actual Size : ');
	errorMessage := concat(errorMessage, UDINT_TO_STRING(SIZEOF(PayloadDataSize)));
	Error(errorMessage);
	RETURN;
END_IF

headerAccessor.UpdateResponseWithSuccess(THIS^);
CompleteResponseWithPayload(PayloadDataAddress, PayloadDataSize);
END_METHOD

METHOD PUBLIC TryGetData : BOOL;
VAR_INPUT
	Destination : REFERENCE TO ResponseData;
END_VAR
IF NOT __ISVALIDREF(Destination) THEN
	RETURN;
END_IF

IF SIZEOF(Destination) <> SIZEOF(responseData) THEN
	RETURN;
END_IF

memcpy(ADR(Destination), ADR(responseData), SIZEOF(Destination));
TryGetData := TRUE;
END_METHOD

END_FUNCTION_BLOCK

// _Internal/Middleware/Stack/MiddlewareStack
{attribute 'linkalways'} 
{attribute 'no_explicit_call' := 'This FB is a CLASS and must be accessed using methods or properties'}
{attribute 'enable_dynamic_creation'}
FUNCTION_BLOCK MiddlewareStack
VAR
	InitialHandler : I_Middleware;
END_VAR

METHOD PUBLIC Handle
VAR_INPUT
	Request : I_Request;
	Response : I_ServerResponse;
END_VAR
IF initialHandler = 0 THEN
	RETURN;
END_IF

initialHandler.Handle(Request, Response);
END_METHOD

METHOD PUBLIC Use
VAR_INPUT
	Handler : I_Middleware;
END_VAR
VAR
	currentHandler : I_Middleware;
END_VAR;
IF initialHandler = 0 THEN
	initialHandler := Handler;
	RETURN;
END_IF

currentHandler := InitialHandler;

WHILE currentHandler.NextMiddleware <> 0 DO
	currentHandler := currentHandler.NextMiddleware;
END_WHILE

currentHandler.NextMiddleware := Handler;
END_METHOD

END_FUNCTION_BLOCK

// _Internal/ResponseId/SequentialResponseIdGenerator
{attribute 'linkalways'} 
{attribute 'no_explicit_call' := 'This FB is a CLASS and must be accessed using methods or properties'}
{attribute 'enable_dynamic_creation'}
FUNCTION_BLOCK SequentialResponseIdGenerator IMPLEMENTS I_ResponseIdGenerator
VAR
	currentCount : UDINT;
END_VAR

METHOD PUBLIC Generate : T_MAXSTRING
VAR_INPUT
END_VAR
currentCount := currentCount + 1;
Generate := UDINT_TO_STRING(currentCount);
END_METHOD

END_FUNCTION_BLOCK

// _Internal/RPC/AsyncRpcCall/AsyncRpcCall
{attribute 'linkalways'} 
{attribute 'no_explicit_call' := 'This FB is a CLASS and must be accessed using methods or properties'}
{attribute 'enable_dynamic_creation'}
{attribute 'TcRpcEnable'}
FUNCTION_BLOCK AsyncRpcCall EXTENDS Disposable IMPLEMENTS I_AsyncRpcCall
VAR
	parameters : I_Deserializer;
	asynchronousRpcResponse : I_AsynchronousRpcResponse;
	handler : I_AsynchronousRpcHandler;
	called : BOOL;
END_VAR

METHOD FB_init : BOOL
VAR_INPUT
	bInitRetains : BOOL; // if TRUE, the retain variables are initialized (warm start / cold start)
	bInCopyCode : BOOL;  // if TRUE, the instance afterwards gets moved into the copy code (online change)
	Parameters : I_Deserializer;
	AsynchronousRpcResponse : I_AsynchronousRpcResponse;
	Handler : I_AsynchronousRpcHandler;
END_VAR
THIS^.parameters := Parameters;
THIS^.asynchronousRpcResponse := AsynchronousRpcResponse;
THIS^.handler := Handler;
END_METHOD

METHOD FB_exit : BOOL
VAR_INPUT
	bInCopyCode : BOOL; // if TRUE, the exit method is called for exiting an instance that is copied afterwards (online change).
END_VAR
IF bInCopyCode THEN
	RETURN;
END_IF

IF called THEN
	RETURN;
END_IF

parameters.Dispose();
asynchronousRpcResponse.RejectWithMessage('RPC : Disposed');
END_METHOD

METHOD PUBLIC Call
VAR_INPUT
END_VAR
IF called THEN 
	RETURN;
END_IF

handler.Handle(parameters, asynchronousRpcResponse);
parameters.Dispose();
called := TRUE;
END_METHOD

END_FUNCTION_BLOCK

// _Internal/RPC/AsyncRpcCall/I_AsyncRpcCall
INTERFACE I_AsyncRpcCall EXTENDS I_Disposable

METHOD PUBLIC Call
VAR_INPUT
END_VAR
END_METHOD

END_INTERFACE

// _Internal/RPC/Response/Async/AsynchronousRpcResponse
{attribute 'linkalways'} 
{attribute 'no_explicit_call' := 'This FB is a CLASS and must be accessed using methods or properties'}
{attribute 'enable_dynamic_creation'}
FUNCTION_BLOCK AsynchronousRpcResponse EXTENDS Disposable IMPLEMENTS I_AsynchronousRpcResponse
VAR
	asyncResponse : I_AsyncResponseSessionData;
	serializer : I_Serializer;
END_VAR

METHOD FB_init : BOOL
VAR_INPUT
	bInitRetains : BOOL; // if TRUE, the retain variables are initialized (warm start / cold start)
	bInCopyCode : BOOL;  // if TRUE, the instance afterwards gets moved into the copy code (online change)
	AsyncResponse : I_AsyncResponseSessionData;
	Serializer : I_Serializer;
END_VAR
THIS^.asyncResponse := AsyncResponse;
THIS^.serializer := Serializer.Clone();
END_METHOD

METHOD FB_exit : BOOL
VAR_INPUT
	bInCopyCode : BOOL; // if TRUE, the exit method is called for exiting an instance that is copied afterwards (online change).
END_VAR
IF bInCopyCode THEN
	RETURN;
END_IF

serializer.Dispose();

IF asyncResponse <> 0 THEN				
	asyncResponse.Dispose();
END_IF
END_METHOD

METHOD PROTECTED SendSuccessResponseUsingSeralizer
VAR_INPUT
	Serializer : I_Serializer;
END_VAR
VAR
	jsonSize : UDINT;
	pJsonString : POINTER TO STRING;
END_VAR
IF asyncResponse = 0 THEN
	RETURN;
END_IF

jsonSize := Serializer.GetSerializedDataLength();

IF jsonSize = 0 THEN
	asyncResponse.Success();
END_IF

pJsonString := __NEW(BYTE, jsonSize);

IF NOT Serializer.TryGetSerializedData(pJsonString, jsonSize) THEN
	asyncResponse.Error('RPC Handler unable to get serialized data');
	__DELETE(pJsonString);
	RETURN;
END_IF

asyncResponse.SuccessWithPayload(pJsonString, jsonSize);
__DELETE(pJsonString);
END_METHOD

METHOD PUBLIC CompleteWithBase64
VAR_INPUT
	pBytes : POINTER TO BYTE;
	nBytes : DINT;
END_VAR
serializer.Reset();
serializer.AddBase64(pBytes, nBytes);
SendSuccessResponseUsingSeralizer(serializer);
Dispose();
END_METHOD

METHOD PUBLIC CompleteWithBool
VAR_INPUT
	Value : BOOL;
END_VAR
serializer.Reset();
serializer.AddBool(Value);
SendSuccessResponseUsingSeralizer(serializer);
Dispose();
END_METHOD

METHOD PUBLIC CompleteWithBytesAsHex
VAR_INPUT
	pBytes : POINTER TO BYTE;
	nBytes : DINT;
END_VAR
serializer.Reset();
serializer.AddBytesAsHex(pBytes, nBytes);
SendSuccessResponseUsingSeralizer(serializer);
Dispose();
END_METHOD

METHOD PUBLIC CompleteWithDateTime
VAR_INPUT
	Value : DATE_AND_TIME;
END_VAR
serializer.Reset();
serializer.AddDateTime(Value);
SendSuccessResponseUsingSeralizer(serializer);
Dispose();
END_METHOD

METHOD PUBLIC CompleteWithDcTime
VAR_INPUT
	Value : DCTIME;
END_VAR
serializer.Reset();
serializer.AddDcTime(Value);
SendSuccessResponseUsingSeralizer(serializer);
Dispose();
END_METHOD

METHOD PUBLIC CompleteWithDint
VAR_INPUT
	Value : DINT;
END_VAR
serializer.Reset();
serializer.AddDint(Value);
SendSuccessResponseUsingSeralizer(serializer);
Dispose();
END_METHOD

METHOD PUBLIC CompleteWithFileTime
VAR_INPUT
	Value : FILETIME;
END_VAR
serializer.Reset();
serializer.AddFileTime(Value);
SendSuccessResponseUsingSeralizer(serializer);
Dispose();
END_METHOD

METHOD PUBLIC CompleteWithLint
VAR_INPUT
	Value : LINT;
END_VAR
serializer.Reset();
serializer.AddLint(Value);
SendSuccessResponseUsingSeralizer(serializer);
Dispose();
END_METHOD

METHOD PUBLIC CompleteWithLreal
VAR_INPUT
	Value : LREAL;
END_VAR
serializer.Reset();
serializer.AddLreal(Value);
SendSuccessResponseUsingSeralizer(serializer);
Dispose();
END_METHOD

METHOD PUBLIC CompleteWithNull
VAR_INPUT
END_VAR
serializer.Reset();
serializer.AddNull();
SendSuccessResponseUsingSeralizer(serializer);
Dispose();
END_METHOD

METHOD PUBLIC CompleteWithObject
VAR_INPUT
	Object : I_Serializable;
END_VAR
serializer.Reset();
Object.SerializeWith(serializer);
SendSuccessResponseUsingSeralizer(serializer);
Dispose();
END_METHOD

METHOD PUBLIC CompleteWithReal
VAR_INPUT
	Value : REAL;
END_VAR
serializer.Reset();
serializer.AddReal(Value);
SendSuccessResponseUsingSeralizer(serializer);
Dispose();
END_METHOD

METHOD PUBLIC CompleteWithSerializer
VAR_INPUT
	Serializer : I_Serializer;
END_VAR
SendSuccessResponseUsingSeralizer(Serializer);
Dispose();
END_METHOD

METHOD PUBLIC CompleteWithString
VAR_INPUT
	Value : T_MAXSTRING;
END_VAR
serializer.Reset();
serializer.AddString(Value);
SendSuccessResponseUsingSeralizer(serializer);
Dispose();
END_METHOD

METHOD PUBLIC CompleteWithUdint
VAR_INPUT
	Value : UDINT;
END_VAR
serializer.Reset();
serializer.AddUdint(Value);
SendSuccessResponseUsingSeralizer(serializer);
Dispose();
END_METHOD

METHOD PUBLIC CompleteWithUlint
VAR_INPUT
	Value : ULINT;
END_VAR
serializer.Reset();
serializer.AddUlint(Value);
SendSuccessResponseUsingSeralizer(serializer);
Dispose();
END_METHOD

METHOD PUBLIC GetSerializer : I_Serializer
VAR_INPUT
END_VAR
GetSerializer := serializer.Clone();
END_METHOD

METHOD PUBLIC RejectWithMessage
VAR_INPUT
	Message : T_MAXSTRING;
END_VAR
IF asyncResponse <> 0 THEN
	asyncResponse.Error(Message);
END_IF

Dispose();
END_METHOD

END_FUNCTION_BLOCK

// _Internal/RPC/Response/Async/I_AsynchronousRpcResponse
INTERFACE I_AsynchronousRpcResponse EXTENDS I_Disposable

METHOD PUBLIC CompleteWithBase64
VAR_INPUT
	pBytes : POINTER TO BYTE;
	nBytes : DINT;
END_VAR
END_METHOD

METHOD PUBLIC CompleteWithBool
VAR_INPUT
	Value : BOOL;
END_VAR
END_METHOD

METHOD PUBLIC CompleteWithBytesAsHex
VAR_INPUT
	pBytes : POINTER TO BYTE;
	nBytes : DINT;
END_VAR
END_METHOD

METHOD PUBLIC CompleteWithDateTime
VAR_INPUT
	Value : DATE_AND_TIME;
END_VAR
END_METHOD

METHOD PUBLIC CompleteWithDcTime
VAR_INPUT
	Value : DCTIME;
END_VAR
END_METHOD

METHOD PUBLIC CompleteWithDint
VAR_INPUT
	Value : DINT;
END_VAR
END_METHOD

METHOD PUBLIC CompleteWithFileTime
VAR_INPUT
	Value : FILETIME;
END_VAR
END_METHOD

METHOD PUBLIC CompleteWithLint
VAR_INPUT
	Value : LINT;
END_VAR
END_METHOD

METHOD PUBLIC CompleteWithLreal
VAR_INPUT
	Value : LREAL;
END_VAR
END_METHOD

METHOD PUBLIC CompleteWithNull
VAR_INPUT
END_VAR
END_METHOD

METHOD PUBLIC CompleteWithObject
VAR_INPUT
	Object : I_Serializable;
END_VAR
END_METHOD

METHOD PUBLIC CompleteWithReal
VAR_INPUT
	Value : REAL;
END_VAR
END_METHOD

METHOD PUBLIC CompleteWithSerializer
VAR_INPUT
	Serializer : I_Serializer;
END_VAR
END_METHOD

METHOD PUBLIC CompleteWithString
VAR_INPUT
	Value : T_MAXSTRING;
END_VAR
END_METHOD

METHOD PUBLIC CompleteWithUdint
VAR_INPUT
	Value : UDINT;
END_VAR
END_METHOD

METHOD PUBLIC CompleteWithUlint
VAR_INPUT
	Value : ULINT;
END_VAR
END_METHOD

METHOD PUBLIC GetSerializer : I_Serializer
VAR_INPUT
END_VAR
END_METHOD

METHOD PUBLIC RejectWithMessage
VAR_INPUT
	Message : T_MAXSTRING;
END_VAR
END_METHOD

END_INTERFACE

// RpcHandler/I_AsynchronousRpcHandler
INTERFACE I_AsynchronousRpcHandler EXTENDS __SYSTEM.IQueryInterface

METHOD Handle
VAR_INPUT
	Parameters : I_Deserializer;
	Response : I_AsynchronousRpcResponse;
END_VAR
END_METHOD

END_INTERFACE

// _Internal/RPC/AsyncRpcCallQueue/AsyncRpcCallQueue
{attribute 'linkalways'} 
{attribute 'no_explicit_call' := 'This FB is a CLASS and must be accessed using methods or properties'}
{attribute 'enable_dynamic_creation'}
{attribute 'TcRpcEnable'}
FUNCTION_BLOCK AsyncRpcCallQueue IMPLEMENTS I_AsyncRpcCallQueue
VAR
	callQueue : Queue;
END_VAR

METHOD FB_exit : BOOL
VAR_INPUT
	bInCopyCode : BOOL; // if TRUE, the exit method is called for exiting an instance that is copied afterwards (online change).
END_VAR
IF bInCopyCode THEN
	RETURN;
END_IF

DisposeAll();
END_METHOD

METHOD PUBLIC CreateCall : I_AsyncRpcCall
VAR_INPUT
	CallingParameters : I_Deserializer;
	CallingAsynchronousRpcResponse : I_AsynchronousRpcResponse;
	CallingHandler : I_AsynchronousRpcHandler;
END_VAR
VAR
	pAsyncRpcCall : POINTER TO AsyncRpcCall;
END_VAR
pAsyncRpcCall := __NEW(AsyncRpcCall(Parameters := CallingParameters, AsynchronousRpcResponse := CallingAsynchronousRpcResponse, Handler := CallingHandler));
CreateCall := pAsyncRpcCall^;
END_METHOD

METHOD PROTECTED DisposeAll
VAR
	asyncRpcCall : I_AsyncRpcCall;
END_VAR
WHILE callQueue.TryDequeue(asyncRpcCall) DO
	asyncRpcCall.Dispose();
END_WHILE
END_METHOD

METHOD PUBLIC CyclicCall
VAR
	asyncRpcCall : I_AsyncRpcCall;
END_VAR
IF callQueue.TryDequeue(asyncRpcCall) THEN
	asyncRpcCall.Call();
	asyncRpcCall.Dispose();
END_IF
END_METHOD

METHOD PUBLIC TryAddRpcCall : BOOL
VAR_INPUT
	CallingParameters : I_Deserializer;
	CallingAsynchronousRpcResponse : I_AsynchronousRpcResponse;
	CallingHandler : I_AsynchronousRpcHandler;
END_VAR
VAR
	asyncRpcCall : I_AsyncRpcCall;
END_VAR
asyncRpcCall := CreateCall(CallingParameters, CallingAsynchronousRpcResponse, CallingHandler);
callQueue.Enqueue(asyncRpcCall);
TryAddRpcCall := TRUE;
END_METHOD

END_FUNCTION_BLOCK

// _Internal/RPC/AsyncRpcCallQueue/I_AsyncRpcCallQueue
INTERFACE I_AsyncRpcCallQueue

METHOD PUBLIC TryAddRpcCall : BOOL
VAR_INPUT
	CallingParameters : I_Deserializer;
	CallingAsynchronousRpcResponse : I_AsynchronousRpcResponse;
	CallingHandler : I_AsynchronousRpcHandler;
END_VAR
END_METHOD

END_INTERFACE

// _Internal/RPC/Handlers/AsynchronousRpcHandlers
{attribute 'linkalways'} 
{attribute 'no_explicit_call' := 'This FB is a CLASS and must be accessed using methods or properties'}
{attribute 'enable_dynamic_creation'}
FUNCTION_BLOCK AsynchronousRpcHandlers IMPLEMENTS I_AsynchronousRpcHandlers, I_HostAsynchronousRpcHandlers
VAR
	handlers : Dictionary;
	_hasHandlers : BOOL;
END_VAR

PROPERTY PUBLIC HasHandlers : BOOL
GET
HasHandlers := _hasHandlers;
END_GET
END_PROPERTY

METHOD PUBLIC RegisterHandler
VAR_INPUT
	MethodName : T_MAXSTRING;
	Handler : I_AsynchronousRpcHandler;
END_VAR
handlers.AddOrUpdate(MethodName, Handler);
_hasHandlers := true;
END_METHOD

METHOD PUBLIC TryGetByMethodName : BOOL
VAR_INPUT
	MethodName : T_MAXSTRING;
	Destination : REFERENCE TO I_AsynchronousRpcHandler;
END_VAR
TryGetByMethodName := handlers.TryGetValue(MethodName, Destination);
END_METHOD

END_FUNCTION_BLOCK

// _Internal/RPC/Handlers/I_AsynchronousRpcHandlers
INTERFACE I_AsynchronousRpcHandlers

PROPERTY PUBLIC HasHandlers : BOOL
GET
END_GET
END_PROPERTY

METHOD PUBLIC TryGetByMethodName : BOOL
VAR_INPUT
	MethodName : T_MAXSTRING;
	Destination : REFERENCE TO I_AsynchronousRpcHandler;
END_VAR
END_METHOD

END_INTERFACE

// _Internal/RPC/Handlers/I_HostAsynchronousRpcHandlers
INTERFACE I_HostAsynchronousRpcHandlers

METHOD PUBLIC RegisterHandler
VAR_INPUT
	MethodName : T_MAXSTRING;
	Handler : I_AsynchronousRpcHandler;
END_VAR
END_METHOD

END_INTERFACE

// _Internal/RPC/Handlers/I_HostSynchronousRpcHandlers
INTERFACE I_HostSynchronousRpcHandlers

METHOD PUBLIC RegisterHandler
VAR_INPUT
	MethodName : T_MAXSTRING;
	Handler : I_SynchronousRpcHandler;
END_VAR
END_METHOD

END_INTERFACE

// RpcHandler/I_SynchronousRpcHandler
INTERFACE I_SynchronousRpcHandler EXTENDS __SYSTEM.IQueryInterface

METHOD Handle
VAR_INPUT
	Parameters : I_Deserializer;
	Response : I_SynchronousRpcResponse;
END_VAR
END_METHOD

END_INTERFACE

// _Internal/RPC/Response/Sync/I_SynchronousRpcResponse
INTERFACE I_SynchronousRpcResponse EXTENDS I_Disposable

METHOD PUBLIC CompleteWithBase64
VAR_INPUT
	pBytes : POINTER TO BYTE;
	nBytes : DINT;
END_VAR
END_METHOD

METHOD PUBLIC CompleteWithBool
VAR_INPUT
	Value : BOOL;
END_VAR
END_METHOD

METHOD PUBLIC CompleteWithBytesAsHex
VAR_INPUT
	pBytes : POINTER TO BYTE;
	nBytes : DINT;
END_VAR
END_METHOD

METHOD PUBLIC CompleteWithDateTime
VAR_INPUT
	Value : DATE_AND_TIME;
END_VAR
END_METHOD

METHOD PUBLIC CompleteWithDcTime
VAR_INPUT
	Value : DCTIME;
END_VAR
END_METHOD

METHOD PUBLIC CompleteWithDint
VAR_INPUT
	Value : DINT;
END_VAR
END_METHOD

METHOD PUBLIC CompleteWithFileTime
VAR_INPUT
	Value : FILETIME;
END_VAR
END_METHOD

METHOD PUBLIC CompleteWithLint
VAR_INPUT
	Value : LINT;
END_VAR
END_METHOD

METHOD PUBLIC CompleteWithLreal
VAR_INPUT
	Value : LREAL;
END_VAR
END_METHOD

METHOD PUBLIC CompleteWithNull
VAR_INPUT
END_VAR
END_METHOD

METHOD PUBLIC CompleteWithObject
VAR_INPUT
	Object : I_Serializable;
END_VAR
END_METHOD

METHOD PUBLIC CompleteWithReal
VAR_INPUT
	Value : REAL;
END_VAR
END_METHOD

METHOD PUBLIC CompleteWithSerializer
VAR_INPUT
	Serializer : I_Serializer;
END_VAR
END_METHOD

METHOD PUBLIC CompleteWithString
VAR_INPUT
	Value : T_MAXSTRING;
END_VAR
END_METHOD

METHOD PUBLIC CompleteWithUdint
VAR_INPUT
	Value : UDINT;
END_VAR
END_METHOD

METHOD PUBLIC CompleteWithUlint
VAR_INPUT
	Value : ULINT;
END_VAR
END_METHOD

METHOD PUBLIC GetSerializer : I_Serializer
VAR_INPUT
END_VAR
END_METHOD

METHOD PUBLIC RejectWithMessage
VAR_INPUT
	Message : T_MAXSTRING;
END_VAR
END_METHOD

METHOD PUBLIC TryMakeAsynchronous : BOOL
VAR_INPUT
	Destination : REFERENCE TO I_AsynchronousRpcResponse;
END_VAR
END_METHOD

END_INTERFACE

// _Internal/RPC/Handlers/I_SynchronousRpcHandlers
INTERFACE I_SynchronousRpcHandlers

PROPERTY PUBLIC HasHandlers : BOOL
GET
END_GET
END_PROPERTY

METHOD PUBLIC TryGetByMethodName : BOOL
VAR_INPUT
	MethodName : T_MAXSTRING;
	Destination : REFERENCE TO I_SynchronousRpcHandler;
END_VAR
END_METHOD

END_INTERFACE

// _Internal/RPC/Handlers/SynchronousRpcHandlers
{attribute 'linkalways'} 
{attribute 'no_explicit_call' := 'This FB is a CLASS and must be accessed using methods or properties'}
{attribute 'enable_dynamic_creation'}
FUNCTION_BLOCK SynchronousRpcHandlers IMPLEMENTS I_SynchronousRpcHandlers, I_HostSynchronousRpcHandlers
VAR
	handlers : Dictionary;
	_hasHandlers : BOOL;
END_VAR

PROPERTY PUBLIC HasHandlers : BOOL
GET
HasHandlers := _hasHandlers;
END_GET
END_PROPERTY

METHOD PUBLIC RegisterHandler
VAR_INPUT
	MethodName : T_MAXSTRING;
	Handler : I_SynchronousRpcHandler;
END_VAR
handlers.AddOrUpdate(MethodName, Handler);
_hasHandlers := true;
END_METHOD

METHOD PUBLIC TryGetByMethodName : BOOL
VAR_INPUT
	MethodName : T_MAXSTRING;
	Destination : REFERENCE TO I_SynchronousRpcHandler;
END_VAR
TryGetByMethodName := handlers.TryGetValue(MethodName, Destination);
END_METHOD

END_FUNCTION_BLOCK

// _Internal/RPC/Manager/I_RpcManager
INTERFACE I_RpcManager

METHOD PUBLIC TryHandleIncomingRequest : BOOL
VAR_INPUT
	Request : I_Request;
	Response : I_ServerResponse;
END_VAR
END_METHOD

END_INTERFACE

// _Internal/RPC/Manager/RpcManager
FUNCTION_BLOCK RpcManager IMPLEMENTS I_RpcManager
VAR
	syncRpcHandlers : I_SynchronousRpcHandlers;
	asyncRpcHandlers : I_AsynchronousRpcHandlers;
	asyncResponseManager : I_AsyncResponseManager;
	headerAccessor : I_RpcHeaderAccessor;
	asyncRpcCallQueue : I_AsyncRpcCallQueue;
END_VAR

METHOD FB_init : BOOL
VAR_INPUT
	bInitRetains : BOOL; // if TRUE, the retain variables are initialized (warm start / cold start)
	bInCopyCode : BOOL;  // if TRUE, the instance afterwards gets moved into the copy code (online change)
	SyncRpcHandlers : I_SynchronousRpcHandlers;
	AsyncRpcHandlers : I_AsynchronousRpcHandlers;
	AsyncResponseManager : I_AsyncResponseManager;
	HeaderAccessor : I_RpcHeaderAccessor;
	AsyncRpcCallQueue : I_AsyncRpcCallQueue;
END_VAR
THIS^.syncRpcHandlers := SyncRpcHandlers;
THIS^.asyncRpcHandlers := AsyncRpcHandlers;
THIS^.asyncResponseManager := AsyncResponseManager;
THIS^.headerAccessor := HeaderAccessor;
THIS^.asyncRpcCallQueue := asyncRpcCallQueue;
END_METHOD

METHOD PROTECTED HandleAsyncRpcRequest
VAR_INPUT
	Request : I_Request;
	Response : I_ServerResponse;
	Handler : I_AsynchronousRpcHandler;
END_VAR
VAR
	deserializer : I_Deserializer;
	serializer : I_Serializer;
	asynchronousRpcResponse : I_AsynchronousRpcResponse;
END_VAR
IF NOT TryCreateSerializer(Request, serializer) THEN
	Response.Error('RPC : Missing or unsupported accept type in header');
	RETURN;
END_IF

IF NOT TryCreateDeserializer(Request, deserializer) THEN
	Response.Error('RPC : Missing or unsupported content type in header');
	serializer.Dispose();
	RETURN;
END_IF

IF NOT TryCreateAsynchronousRpcResponse(Response, serializer, asynchronousRpcResponse) THEN
	Response.Error('RPC : Unable to create asynchronous response for handler');
	serializer.Dispose();
	deserializer.Dispose();
	RETURN;
END_IF

IF NOT asyncRpcCallQueue.TryAddRpcCall(deserializer, asynchronousRpcResponse, Handler) THEN
	serializer.Dispose();
	deserializer.Dispose();
	asynchronousRpcResponse.RejectWithMessage('RPC : Unable to create rpc call');
	RETURN;
END_IF

// we can dispose of the serializer at this stage as it was only used as a prototype.
// this is because when the asynchronousRpcResponse is created then it clones it's serializer. 
serializer.Dispose();
END_METHOD

METHOD PROTECTED HandleSyncRpcRequest
VAR_INPUT
	Request : I_Request;
	Response : I_ServerResponse;
	Handler : I_SynchronousRpcHandler;
END_VAR
VAR
	deserializer : I_Deserializer;
	serializer : I_Serializer;
	synchronousRpcResponse : I_SynchronousRpcResponse;
END_VAR
IF NOT TryCreateSerializer(Request, serializer) THEN
	Response.Error('RPC : Missing or unsupported accept type in header');
	RETURN;
END_IF

IF NOT TryCreateDeserializer(Request, deserializer) THEN
	Response.Error('RPC : Missing or unsupported content type in header');
	serializer.Dispose();
	RETURN;
END_IF

IF NOT TryCreateSynchronousRpcResponse(Response, serializer, synchronousRpcResponse) THEN
	Response.Error('RPC : Unable to create synchronous response for handler');
	serializer.Dispose();
	deserializer.Dispose();
	RETURN;
END_IF

Handler.Handle(deserializer, synchronousRpcResponse);

synchronousRpcResponse.Dispose();
deserializer.Dispose();
serializer.Dispose();

IF NOT Response.HeadersSent THEN
	Response.Error('RPC : Handler did not return a valid response');
	RETURN;
END_IF
END_METHOD

METHOD PROTECTED TryCreateAsynchronousRpcResponse : BOOL
VAR_INPUT
	Response : I_ServerResponse;
	ResponseSerializer : I_Serializer;
	Destination : REFERENCE TO I_AsynchronousRpcResponse;
END_VAR
VAR
	asynchronousRpcResponseFactory : AsynchronousRpcResponseFactory(Response, ResponseSerializer, asyncResponseManager);
END_VAR
IF Response = 0 THEN 
	RETURN;
END_IF

IF ResponseSerializer = 0 THEN
	RETURN;
END_IF

TryCreateAsynchronousRpcResponse := asynchronousRpcResponseFactory.TryCreate(Destination);
END_METHOD

METHOD PROTECTED TryCreateDeserializer : BOOL
VAR_INPUT
	Request : I_Request;
	Destination : REFERENCE TO I_Deserializer;
END_VAR
VAR
	contentType : T_MAXSTRING;
	pJsonDeserializer : POINTER TO JsonDeserializer;
	pJson : POINTER TO STRING;
END_VAR
IF NOT(headerAccessor.TryGetContentTypeFromRequest(Request, contentType)) THEN
	// unlike TryCreateSerializer, a content type must be included.  Therefore if it 
	// is missing a fault will be raised and the request will be rejected.
	RETURN;
END_IF

IF contentType = headerAccessor.ContentType_Json THEN
	pJsonDeserializer := __NEW(JsonDeserializer);
	pJson := request.PayloadAddress;
	pJsonDeserializer^.TryLoad(pJson^);
	
	Destination := pJsonDeserializer^;
	TryCreateDeserializer := TRUE;
	RETURN;
END_IF

// add other supported formats here...
END_METHOD

METHOD PROTECTED TryCreateSerializer : BOOL
VAR_INPUT
	Request : I_Request;
	Destination : REFERENCE TO I_Serializer;
END_VAR
VAR
	acceptType : T_MAXSTRING;
	pJsonSerializer : POINTER TO JsonSerializer;
END_VAR
IF NOT(headerAccessor.TryGetAcceptResponseFormatFromRequest(Request, acceptType)) THEN
	// if no header is provided for the accept type, then the line below selects the default return type. 
	// change this line to change the default.
	acceptType := headerAccessor.ContentType_Json;
END_IF

IF acceptType = headerAccessor.ContentType_Json THEN
	pJsonSerializer := __NEW(JsonSerializer);
	Destination := pJsonSerializer^;
	TryCreateSerializer := TRUE;
	RETURN;
END_IF

// add other supported formats here...
END_METHOD

METHOD PROTECTED TryCreateSynchronousRpcResponse : BOOL
VAR_INPUT
	Response : I_ServerResponse;
	ResponseSerializer : I_Serializer;
	Destination : REFERENCE TO I_SynchronousRpcResponse;
END_VAR
VAR
	pSynchronousRpcResponse : POINTER TO SynchronousRpcResponse;
END_VAR
IF Response = 0 THEN 
	RETURN;
END_IF

IF ResponseSerializer = 0 THEN
	RETURN;
END_IF

pSynchronousRpcResponse := __NEW(SynchronousRpcResponse(ServerResponse := Response, Serializer := ResponseSerializer, AsyncResponseManager := THIS^.asyncResponseManager));
Destination := pSynchronousRpcResponse^;
TryCreateSynchronousRpcResponse := TRUE;
END_METHOD

METHOD PUBLIC TryHandleIncomingRequest : BOOL
VAR_INPUT
	Request : I_Request;
	Response : I_ServerResponse;
END_VAR
VAR
	requestType : T_MAXSTRING;
	methodName : T_MAXSTRING;
	asyncRpcHandler : I_AsynchronousRpcHandler;
	syncRpcHandler : I_SynchronousRpcHandler;
END_VAR
IF NOT headerAccessor.TryGetTypeFromRequest(Request, requestType) THEN
	RETURN;
END_IF

IF requestType <> 'RPC 1.0' THEN
	RETURN;
END_IF

IF NOT headerAccessor.TryGetMethodNameFromRequest(Request, methodName) THEN
	Response.Error('RPC : Missing RPC method name');
	TryHandleIncomingRequest := TRUE;
	RETURN;
END_IF

IF asyncRpcHandlers.hasHandlers AND_THEN asyncRpcHandlers.TryGetByMethodName(methodName, asyncRpcHandler) THEN
	HandleAsyncRpcRequest(Request, Response, asyncRpcHandler);
	TryHandleIncomingRequest := TRUE;
	RETURN;
END_IF

IF syncRpcHandlers.hasHandlers AND_THEN syncRpcHandlers.TryGetByMethodName(methodName, syncRpcHandler) THEN
	HandleSyncRpcRequest(Request, Response, syncRpcHandler);
	TryHandleIncomingRequest := TRUE;
	RETURN;
END_IF
END_METHOD

END_FUNCTION_BLOCK

// _Internal/RPC/Response/Sync/SynchronousRpcResponse
{attribute 'linkalways'} 
{attribute 'no_explicit_call' := 'This FB is a CLASS and must be accessed using methods or properties'}
{attribute 'enable_dynamic_creation'}
FUNCTION_BLOCK SynchronousRpcResponse EXTENDS Disposable IMPLEMENTS I_SynchronousRpcResponse
VAR
	serverResponse : I_ServerResponse;
	serializer : I_Serializer;
	asyncResponseManager : I_AsyncResponseManager;
END_VAR

METHOD FB_init : BOOL
VAR_INPUT
	bInitRetains : BOOL; // if TRUE, the retain variables are initialized (warm start / cold start)
	bInCopyCode : BOOL;  // if TRUE, the instance afterwards gets moved into the copy code (online change)
	ServerResponse : I_ServerResponse;
	Serializer : I_Serializer;
	AsyncResponseManager : I_AsyncResponseManager;
END_VAR
THIS^.serverResponse := ServerResponse;
THIS^.serializer := Serializer.Clone();
THIS^.asyncResponseManager := AsyncResponseManager;
END_METHOD

METHOD FB_exit : BOOL
VAR_INPUT
	bInCopyCode : BOOL; // if TRUE, the exit method is called for exiting an instance that is copied afterwards (online change).
END_VAR
IF bInCopyCode THEN
	RETURN;
END_IF

serializer.Dispose();
END_METHOD

METHOD PROTECTED SendSuccessResponseUsingSeralizer
VAR_INPUT
	Serializer : I_Serializer;
END_VAR
VAR
	jsonSize : UDINT;
	pJsonString : POINTER TO STRING;
END_VAR
jsonSize := Serializer.GetSerializedDataLength();

IF jsonSize = 0 THEN
	serverResponse.Success();
END_IF

pJsonString := __NEW(BYTE, jsonSize);

IF NOT Serializer.TryGetSerializedData(pJsonString, jsonSize) THEN
	serverResponse.Error('RPC Handler unable to get serialized data');
	__DELETE(pJsonString);
	RETURN;
END_IF

serverResponse.SuccessWithPayload(pJsonString, jsonSize);
__DELETE(pJsonString);
END_METHOD

METHOD PUBLIC CompleteWithBase64
VAR_INPUT
	pBytes : POINTER TO BYTE;
	nBytes : DINT;
END_VAR
serializer.Reset();
serializer.AddBase64(pBytes, nBytes);
SendSuccessResponseUsingSeralizer(serializer);
END_METHOD

METHOD PUBLIC CompleteWithBool
VAR_INPUT
	Value : BOOL;
END_VAR
serializer.Reset();
serializer.AddBool(Value);
SendSuccessResponseUsingSeralizer(serializer);
END_METHOD

METHOD PUBLIC CompleteWithBytesAsHex
VAR_INPUT
	pBytes : POINTER TO BYTE;
	nBytes : DINT;
END_VAR
serializer.Reset();
serializer.AddBytesAsHex(pBytes, nBytes);
SendSuccessResponseUsingSeralizer(serializer);
END_METHOD

METHOD PUBLIC CompleteWithDateTime
VAR_INPUT
	Value : DATE_AND_TIME;
END_VAR
serializer.Reset();
serializer.AddDateTime(Value);
SendSuccessResponseUsingSeralizer(serializer);
END_METHOD

METHOD PUBLIC CompleteWithDcTime
VAR_INPUT
	Value : DCTIME;
END_VAR
serializer.Reset();
serializer.AddDcTime(Value);
SendSuccessResponseUsingSeralizer(serializer);
END_METHOD

METHOD PUBLIC CompleteWithDint
VAR_INPUT
	Value : DINT;
END_VAR
serializer.Reset();
serializer.AddDint(Value);
SendSuccessResponseUsingSeralizer(serializer);
END_METHOD

METHOD PUBLIC CompleteWithFileTime
VAR_INPUT
	Value : FILETIME;
END_VAR
serializer.Reset();
serializer.AddFileTime(Value);
SendSuccessResponseUsingSeralizer(serializer);
END_METHOD

METHOD PUBLIC CompleteWithLint
VAR_INPUT
	Value : LINT;
END_VAR
serializer.Reset();
serializer.AddLint(Value);
SendSuccessResponseUsingSeralizer(serializer);
END_METHOD

METHOD PUBLIC CompleteWithLreal
VAR_INPUT
	Value : LREAL;
END_VAR
serializer.Reset();
serializer.AddLreal(Value);
SendSuccessResponseUsingSeralizer(serializer);
END_METHOD

METHOD PUBLIC CompleteWithNull
VAR_INPUT
END_VAR
serializer.Reset();
serializer.AddNull();
SendSuccessResponseUsingSeralizer(serializer);
END_METHOD

METHOD PUBLIC CompleteWithObject
VAR_INPUT
	Object : I_Serializable;
END_VAR
serializer.Reset();
Object.SerializeWith(serializer);
SendSuccessResponseUsingSeralizer(serializer);
END_METHOD

METHOD PUBLIC CompleteWithReal
VAR_INPUT
	Value : REAL;
END_VAR
serializer.Reset();
serializer.AddReal(Value);
SendSuccessResponseUsingSeralizer(serializer);
END_METHOD

METHOD PUBLIC CompleteWithSerializer
VAR_INPUT
	Serializer : I_Serializer;
END_VAR
SendSuccessResponseUsingSeralizer(Serializer);
END_METHOD

METHOD PUBLIC CompleteWithString
VAR_INPUT
	Value : T_MAXSTRING;
END_VAR
serializer.Reset();
serializer.AddString(Value);
SendSuccessResponseUsingSeralizer(serializer);
END_METHOD

METHOD PUBLIC CompleteWithUdint
VAR_INPUT
	Value : UDINT;
END_VAR
serializer.Reset();
serializer.AddUdint(Value);
SendSuccessResponseUsingSeralizer(serializer);
END_METHOD

METHOD PUBLIC CompleteWithUlint
VAR_INPUT
	Value : ULINT;
END_VAR
serializer.Reset();
serializer.AddUlint(Value);
SendSuccessResponseUsingSeralizer(serializer);
END_METHOD

METHOD PUBLIC GetSerializer : I_Serializer
VAR_INPUT
END_VAR
GetSerializer := serializer.Clone();
END_METHOD

METHOD PUBLIC RejectWithMessage
VAR_INPUT
	Message : T_MAXSTRING;
END_VAR
serverResponse.Error(Message);
END_METHOD

METHOD PUBLIC TryMakeAsynchronous : BOOL
VAR_INPUT
	Destination : REFERENCE TO I_AsynchronousRpcResponse;
END_VAR
VAR
	asynchronousRpcResponseFactory : AsynchronousRpcResponseFactory(serverResponse, serializer, asyncResponseManager);
END_VAR
TryMakeAsynchronous := asynchronousRpcResponseFactory.TryCreate(Destination);
END_METHOD

END_FUNCTION_BLOCK

// _Internal/RPC/Response/Factory/AsynchronousRpcResponseFactory
{attribute 'linkalways'} 
{attribute 'no_explicit_call' := 'This FB is a CLASS and must be accessed using methods or properties'}
{attribute 'enable_dynamic_creation'}
FUNCTION_BLOCK AsynchronousRpcResponseFactory IMPLEMENTS I_AsynchronousRpcResponseFactory
VAR
	serverResponse : I_ServerResponse;
	serializer : I_Serializer;
	asyncResponseManager : I_AsyncResponseManager;
END_VAR

